LIN {X 0,Y 360.744,Z 841.948,A -85,B 0,C 180,E1 -13041.597,E2 -13041.597} C_VEL
LIN {X 0,Y 360.57,Z 846.721,A -85,B 0,C 180,E1 -13043.283,E2 -13043.283} C_VEL
LIN {X 0,Y 360.444,Z 850.328,A -85,B 0,C 180,E1 -13044.965,E2 -13044.965} C_VEL
LIN {X 0,Y 360.392,Z 852.877,A -85,B 0,C 180,E1 -13046.645,E2 -13046.645} C_VEL
LIN {X 0,Y 360.505,Z 854.049,A -85,B 0,C 180,E1 -13047.764,E2 -13047.764} C_VEL
LIN {X 0,Y 360.532,Z 854.752,A -85,B 0,C 180,E1 -13048.882,E2 -13048.882} C_VEL
LIN {X 0,Y 360.519,Z 855.046,A -85,B 0,C 180,E1 -13049.999,E2 -13049.999} C_VEL
LIN {X 0,Y 360.53,Z 854.935,A -85,B 0,C 180,E1 -13051.116,E2 -13051.116} C_VEL
LIN {X 0,Y 360.472,Z 854.395,A -85,B 0,C 180,E1 -13052.233,E2 -13052.233} C_VEL
LIN {X 0,Y 360.384,Z 853.407,A -85,B 0,C 180,E1 -13053.353,E2 -13053.353} C_VEL
LIN {X 0,Y 360.41,Z 852.013,A -85,B 0,C 180,E1 -13054.472,E2 -13054.472} C_VEL
LIN {X 0,Y 360.39,Z 849.445,A -85,B 0,C 180,E1 -13055.978,E2 -13055.978} C_VEL
LIN {X 0,Y 360.645,Z 845.108,A -85,B 0,C 180,E1 -13057.839,E2 -13057.839} C_VEL
LIN {X 0,Y 360.987,Z 839.985,A -85,B 0,C 180,E1 -13059.524,E2 -13059.524} C_VEL
LIN {X 0,Y 361.519,Z 833.569,A -85,B 0,C 180,E1 -13061.208,E2 -13061.208} C_VEL
LIN {X 0,Y 362.453,Z 825.598,A -85,B 0,C 180,E1 -13062.883,E2 -13062.883} C_VEL
LIN {X 0,Y 363.304,Z 817.472,A -85,B 0,C 180,E1 -13064.278,E2 -13064.278} C_VEL
LIN {X 0,Y 364.433,Z 806.509,A -85,B 0,C 180,E1 -13065.806,E2 -13065.806} C_VEL
LIN {X 0,Y 365.658,Z 795.285,A -85,B 0,C 180,E1 -13067.043,E2 -13067.043} C_VEL
LIN {X 0,Y 366.98,Z 782.593,A -85,B 0,C 180,E1 -13068.13,E2 -13068.13} C_VEL
LIN {X 0,Y 367.909,Z 771.311,A -85,B 0,C 180,E1 -13068.876,E2 -13068.876} C_VEL
LIN {X 0,Y 368.869,Z 757.948,A -85,B 0,C 180,E1 -13069.512,E2 -13069.512} C_VEL
LIN {X 0,Y 369.409,Z 745.082,A -85,B 0,C 180,E1 -13069.916,E2 -13069.916} C_VEL
LIN {X 0,Y 371,Z 678.071,A -85,B 0,C 180,E1 -13071.407,E2 -13071.407} C_VEL
LIN {X 0,Y 368.045,Z 656.105,A -85,B 0,C 180,E1 -13072.161,E2 -13072.161} C_VEL
LIN {X 0,Y 365.134,Z 639.929,A -85,B 0,C 180,E1 -13072.806,E2 -13072.806} C_VEL
LIN {X 0,Y 366.915,Z 623.577,A -85,B 0,C 180,E1 -13076.443,E2 -13076.443} C_VEL
LIN {X 0,Y 365.233,Z 614.506,A -85,B 0,C 180,E1 -13078.753,E2 -13078.753} C_VEL
LIN {X 0,Y 362.83,Z 604.307,A -85,B 0,C 180,E1 -13081.539,E2 -13081.539} C_VEL
LIN {X 0,Y 361.863,Z 600.413,A -85,B 0,C 180,E1 -13082.693,E2 -13082.693} C_VEL
LIN {X 0,Y 361.865,Z 600.411,A -85,B 0,C 180,E1 -13085.635,E2 -13085.635} C_VEL
LIN {X 0,Y 361.871,Z 600.411,A -85,B 0,C 180,E1 -13089.026,E2 -13089.026} C_VEL
LIN {X 0,Y 361.853,Z 600.414,A -85,B 0,C 180,E1 -13092.434,E2 -13092.434} C_VEL
LIN {X 0,Y 361.908,Z 600.407,A -85,B 0,C 180,E1 -13095.93,E2 -13095.93} C_VEL
LIN {X 0,Y 361.9,Z 600.405,A -85,B 0,C 180,E1 -13099.231,E2 -13099.231} C_VEL
LIN {X 0,Y 361.868,Z 600.406,A -85,B 0,C 180,E1 -13102.982,E2 -13102.982} C_VEL
LIN {X 0,Y 361.857,Z 600.409,A -85,B 0,C 180,E1 -13106.628,E2 -13106.628} C_VEL
LIN {X 0,Y 361.872,Z 600.405,A -85,B 0,C 180,E1 -13109.672,E2 -13109.672} C_VEL
LIN {X 0,Y 361.947,Z 600.394,A -85,B 0,C 180,E1 -13113.474,E2 -13113.474} C_VEL
LIN {X 0,Y 361.884,Z 600.404,A -85,B 0,C 180,E1 -13117.144,E2 -13117.144} C_VEL
LIN {X 0,Y 361.913,Z 600.405,A -85,B 0,C 180,E1 -13120.724,E2 -13120.724} C_VEL
LIN {X 0,Y 361.938,Z 600.402,A -85,B 0,C 180,E1 -13124.226,E2 -13124.226} C_VEL
LIN {X 0,Y 361.992,Z 600.395,A -85,B 0,C 180,E1 -13126.527,E2 -13126.527} C_VEL
LIN {X 0,Y 362.028,Z 600.388,A -85,B 0,C 180,E1 -13129.938,E2 -13129.938} C_VEL
LIN {X 0,Y 362.142,Z 600.375,A -85,B 0,C 180,E1 -13132.192,E2 -13132.192} C_VEL
LIN {X 0,Y 362.11,Z 600.379,A -85,B 0,C 180,E1 -13134.431,E2 -13134.431} C_VEL
LIN {X 0,Y 362.275,Z 600.359,A -85,B 0,C 180,E1 -13137.776,E2 -13137.776} C_VEL
LIN {X 0,Y 362.421,Z 600.343,A -85,B 0,C 180,E1 -13140,E2 -13140} C_VEL
LIN {X 0,Y 362.275,Z 600.359,A -85,B 0,C 180,E1 -13142.223,E2 -13142.223} C_VEL
LIN {X 0,Y 362.17,Z 600.377,A -85,B 0,C 180,E1 -13146.686,E2 -13146.686} C_VEL
LIN {X 0,Y 362.067,Z 600.387,A -85,B 0,C 180,E1 -13148.933,E2 -13148.933} C_VEL
LIN {X 0,Y 362.037,Z 600.45,A -85,B 0,C 180,E1 -13150.274,E2 -13150.274} C_VEL
LIN {X 0,Y 363.166,Z 605.77,A -85,B 0,C 180,E1 -13152.113,E2 -13152.113} C_VEL
LIN {X 0,Y 370.828,Z 623.781,A -85,B 0,C 180,E1 -13153.202,E2 -13153.202} C_VEL
LIN {X 0,Y 372.101,Z 628.288,A -85,B 0,C 180,E1 -13153.409,E2 -13153.409} C_VEL
LIN {X 0,Y 369.856,Z 712.137,A -85,B 0,C 180,E1 -13155.306,E2 -13155.306} C_VEL
LIN {X 0,Y 369.281,Z 725.643,A -85,B 0,C 180,E1 -13155.842,E2 -13155.842} C_VEL
LIN {X 0,Y 368.533,Z 737.945,A -85,B 0,C 180,E1 -13156.55,E2 -13156.55} C_VEL
LIN {X 0,Y 367.596,Z 750.201,A -85,B 0,C 180,E1 -13157.507,E2 -13157.507} C_VEL
LIN {X 0,Y 366.603,Z 761.038,A -85,B 0,C 180,E1 -13158.585,E2 -13158.585} C_VEL
LIN {X 0,Y 365.372,Z 771.583,A -85,B 0,C 180,E1 -13159.891,E2 -13159.891} C_VEL
LIN {X 0,Y 364.418,Z 780.085,A -85,B 0,C 180,E1 -13161.199,E2 -13161.199} C_VEL
LIN {X 0,Y 363.405,Z 788.357,A -85,B 0,C 180,E1 -13162.755,E2 -13162.755} C_VEL
LIN {X 0,Y 362.543,Z 795.203,A -85,B 0,C 180,E1 -13164.345,E2 -13164.345} C_VEL
LIN {X 0,Y 361.987,Z 800.581,A -85,B 0,C 180,E1 -13165.902,E2 -13165.902} C_VEL
LIN {X 0,Y 361.349,Z 805.776,A -85,B 0,C 180,E1 -13167.826,E2 -13167.826} C_VEL
LIN {X 0,Y 360.895,Z 809.537,A -85,B 0,C 180,E1 -13169.774,E2 -13169.774} C_VEL
LIN {X 0,Y 360.552,Z 812.009,A -85,B 0,C 180,E1 -13171.755,E2 -13171.755} C_VEL
LIN {X 0,Y 360.407,Z 812.942,A -85,B 0,C 180,E1 -13173.093,E2 -13173.093} C_VEL
LIN {X 0,Y 360.341,Z 813.24,A -85,B 0,C 180,E1 -13175.002,E2 -13175.002} C_VEL
LIN {X 0,Y 360.356,Z 812.132,A -85,B 0,C 180,E1 -13177.199,E2 -13177.199} C_VEL
LIN {X 0,Y 360.585,Z 809.482,A -85,B 0,C 180,E1 -13179.344,E2 -13179.344} C_VEL
LIN {X 0,Y 360.805,Z 807.257,A -85,B 0,C 180,E1 -13180.567,E2 -13180.567} C_VEL
LIN {X 0,Y 361.082,Z 803.145,A -85,B 0,C 180,E1 -13182.303,E2 -13182.303} C_VEL
LIN {X 0,Y 361.548,Z 797.876,A -85,B 0,C 180,E1 -13184.011,E2 -13184.011} C_VEL
LIN {X 0,Y 362.233,Z 790.465,A -85,B 0,C 180,E1 -13185.879,E2 -13185.879} C_VEL
LIN {X 0,Y 363.055,Z 782.045,A -85,B 0,C 180,E1 -13187.563,E2 -13187.563} C_VEL
LIN {X 0,Y 363.939,Z 772.774,A -85,B 0,C 180,E1 -13189.051,E2 -13189.051} C_VEL
LIN {X 0,Y 364.878,Z 762.379,A -85,B 0,C 180,E1 -13190.394,E2 -13190.394} C_VEL
LIN {X 0,Y 365.792,Z 751.243,A -85,B 0,C 180,E1 -13191.55,E2 -13191.55} C_VEL
LIN {X 0,Y 366.608,Z 739.771,A -85,B 0,C 180,E1 -13192.481,E2 -13192.481} C_VEL
LIN {X 0,Y 367.297,Z 726.855,A -85,B 0,C 180,E1 -13193.278,E2 -13193.278} C_VEL
LIN {X 0,Y 367.781,Z 714.021,A -85,B 0,C 180,E1 -13193.836,E2 -13193.836} C_VEL
LIN {X 0,Y 368.178,Z 697.844,A -85,B 0,C 180,E1 -13194.249,E2 -13194.249} C_VEL
LIN {X 0,Y 369.593,Z 625.625,A -85,B 0,C 180,E1 -13195.797,E2 -13195.797} C_VEL
LIN {X 0,Y 367.76,Z 618.455,A -85,B 0,C 180,E1 -13196.058,E2 -13196.058} C_VEL
LIN {X 0,Y 362.366,Z 602.699,A -85,B 0,C 180,E1 -13196.733,E2 -13196.733} C_VEL
LIN {X 0,Y 361.879,Z 600.408,A -85,B 0,C 180,E1 -13197.473,E2 -13197.473} C_VEL
LIN {X 0,Y 361.896,Z 600.402,A -85,B 0,C 180,E1 -13200.956,E2 -13200.956} C_VEL
LIN {X 0,Y 361.951,Z 600.396,A -85,B 0,C 180,E1 -13203.476,E2 -13203.476} C_VEL
LIN {X 0,Y 361.891,Z 600.402,A -85,B 0,C 180,E1 -13207.146,E2 -13207.146} C_VEL
LIN {X 0,Y 361.926,Z 600.399,A -85,B 0,C 180,E1 -13210.726,E2 -13210.726} C_VEL
LIN {X 0,Y 361.945,Z 600.402,A -85,B 0,C 180,E1 -13214.227,E2 -13214.227} C_VEL
LIN {X 0,Y 361.999,Z 600.393,A -85,B 0,C 180,E1 -13216.529,E2 -13216.529} C_VEL
LIN {X 0,Y 362.036,Z 600.387,A -85,B 0,C 180,E1 -13219.939,E2 -13219.939} C_VEL
LIN {X 0,Y 362.152,Z 600.374,A -85,B 0,C 180,E1 -13222.194,E2 -13222.194} C_VEL
LIN {X 0,Y 362.119,Z 600.381,A -85,B 0,C 180,E1 -13224.433,E2 -13224.433} C_VEL
LIN {X 0,Y 362.284,Z 600.354,A -85,B 0,C 180,E1 -13227.778,E2 -13227.778} C_VEL
LIN {X 0,Y 362.427,Z 600.337,A -85,B 0,C 180,E1 -13230.001,E2 -13230.001} C_VEL
LIN {X 0,Y 362.284,Z 600.356,A -85,B 0,C 180,E1 -13232.225,E2 -13232.225} C_VEL
LIN {X 0,Y 362.174,Z 600.374,A -85,B 0,C 180,E1 -13236.687,E2 -13236.687} C_VEL
LIN {X 0,Y 362.034,Z 600.385,A -85,B 0,C 180,E1 -13239.616,E2 -13239.616} C_VEL
LIN {X 0,Y 361.354,Z 600.474,A -85,B 0,C 180,E1 -13240.544,E2 -13240.544} C_VEL
LIN {X 0,Y 358.482,Z 600.827,A -85,B 0,C 180,E1 -13242.053,E2 -13242.053} C_VEL
LIN {X 0,Y 356.053,Z 601.131,A -85,B 0,C 180,E1 -13243.274,E2 -13243.274} C_VEL
LIN {X 0,Y 355.008,Z 601.261,A -85,B 0,C 180,E1 -13244.219,E2 -13244.219} C_VEL
LIN {X 0,Y 354.921,Z 601.273,A -85,B 0,C 180,E1 -13244.539,E2 -13244.539} C_VEL
LIN {X 0,Y 354.904,Z 601.275,A -85,B 0,C 180,E1 -13248.473,E2 -13248.473} C_VEL
LIN {X 0,Y 354.838,Z 601.281,A -85,B 0,C 180,E1 -13252.107,E2 -13252.107} C_VEL
LIN {X 0,Y 354.902,Z 601.273,A -85,B 0,C 180,E1 -13255.828,E2 -13255.828} C_VEL
LIN {X 0,Y 354.821,Z 601.284,A -85,B 0,C 180,E1 -13259.683,E2 -13259.683} C_VEL
LIN {X 0,Y 354.81,Z 601.286,A -85,B 0,C 180,E1 -13263.703,E2 -13263.703} C_VEL
LIN {X 0,Y 354.801,Z 601.286,A -85,B 0,C 180,E1 -13266.46,E2 -13266.46} C_VEL
LIN {X 0,Y 354.828,Z 601.287,A -85,B 0,C 180,E1 -13269.424,E2 -13269.424} C_VEL
LIN {X 0,Y 354.792,Z 601.289,A -85,B 0,C 180,E1 -13272.868,E2 -13272.868} C_VEL
LIN {X 0,Y 354.784,Z 601.288,A -85,B 0,C 180,E1 -13276.106,E2 -13276.106} C_VEL
LIN {X 0,Y 354.792,Z 601.29,A -85,B 0,C 180,E1 -13279.18,E2 -13279.18} C_VEL
LIN {X 0,Y 354.811,Z 601.284,A -85,B 0,C 180,E1 -13282.403,E2 -13282.403} C_VEL
LIN {X 0,Y 354.817,Z 601.285,A -85,B 0,C 180,E1 -13284.941,E2 -13284.941} C_VEL
LIN {X 0,Y 354.8,Z 601.286,A -85,B 0,C 180,E1 -13288.405,E2 -13288.405} C_VEL
LIN {X 0,Y 354.856,Z 601.285,A -85,B 0,C 180,E1 -13291.62,E2 -13291.62} C_VEL
LIN {X 0,Y 354.904,Z 601.275,A -85,B 0,C 180,E1 -13294.173,E2 -13294.173} C_VEL
LIN {X 0,Y 354.821,Z 601.289,A -85,B 0,C 180,E1 -13297.893,E2 -13297.893} C_VEL
LIN {X 0,Y 354.928,Z 601.276,A -85,B 0,C 180,E1 -13301.892,E2 -13301.892} C_VEL
LIN {X 0,Y 354.949,Z 601.273,A -85,B 0,C 180,E1 -13305.981,E2 -13305.981} C_VEL
LIN {X 0,Y 354.983,Z 601.266,A -85,B 0,C 180,E1 -13309.736,E2 -13309.736} C_VEL
LIN {X 0,Y 355.13,Z 601.245,A -85,B 0,C 180,E1 -13313.181,E2 -13313.181} C_VEL
LIN {X 0,Y 355.249,Z 601.232,A -85,B 0,C 180,E1 -13317.733,E2 -13317.733} C_VEL
LIN {X 0,Y 355.402,Z 601.215,A -85,B 0,C 180,E1 -13320,E2 -13320} C_VEL
LIN {X 0,Y 355.249,Z 601.236,A -85,B 0,C 180,E1 -13322.268,E2 -13322.268} C_VEL
LIN {X 0,Y 355.132,Z 601.246,A -85,B 0,C 180,E1 -13326.819,E2 -13326.819} C_VEL
LIN {X 0,Y 354.984,Z 601.268,A -85,B 0,C 180,E1 -13330.264,E2 -13330.264} C_VEL
LIN {X 0,Y 354.949,Z 601.269,A -85,B 0,C 180,E1 -13334.019,E2 -13334.019} C_VEL
LIN {X 0,Y 354.896,Z 601.276,A -85,B 0,C 180,E1 -13338.092,E2 -13338.092} C_VEL
LIN {X 0,Y 354.823,Z 601.285,A -85,B 0,C 180,E1 -13342.107,E2 -13342.107} C_VEL
LIN {X 0,Y 354.905,Z 601.273,A -85,B 0,C 180,E1 -13345.827,E2 -13345.827} C_VEL
LIN {X 0,Y 354.86,Z 601.278,A -85,B 0,C 180,E1 -13349.678,E2 -13349.678} C_VEL
LIN {X 0,Y 354.812,Z 601.284,A -85,B 0,C 180,E1 -13353.702,E2 -13353.702} C_VEL
LIN {X 0,Y 354.803,Z 601.288,A -85,B 0,C 180,E1 -13356.459,E2 -13356.459} C_VEL
LIN {X 0,Y 354.83,Z 601.284,A -85,B 0,C 180,E1 -13359.423,E2 -13359.423} C_VEL
LIN {X 0,Y 354.794,Z 601.292,A -85,B 0,C 180,E1 -13362.867,E2 -13362.867} C_VEL
LIN {X 0,Y 354.78,Z 601.288,A -85,B 0,C 180,E1 -13366.104,E2 -13366.104} C_VEL
LIN {X 0,Y 354.794,Z 601.292,A -85,B 0,C 180,E1 -13369.179,E2 -13369.179} C_VEL
LIN {X 0,Y 354.813,Z 601.284,A -85,B 0,C 180,E1 -13372.402,E2 -13372.402} C_VEL
LIN {X 0,Y 354.817,Z 601.287,A -85,B 0,C 180,E1 -13374.94,E2 -13374.94} C_VEL
LIN {X 0,Y 354.846,Z 601.486,A -85,B 0,C 180,E1 -13378.51,E2 -13378.51} C_VEL
LIN {X 0,Y 357.812,Z 615.009,A -85,B 0,C 180,E1 -13381.874,E2 -13381.874} C_VEL
LIN {X 0,Y 359.157,Z 622.011,A -85,B 0,C 180,E1 -13383.553,E2 -13383.553} C_VEL
LIN {X 0,Y 358.818,Z 627.547,A -85,B 0,C 180,E1 -13384.784,E2 -13384.784} C_VEL
LIN {X 0,Y 357.382,Z 642.401,A -85,B 0,C 180,E1 -13387.999,E2 -13387.999} C_VEL
LIN {X 0,Y 362.247,Z 679.252,A -85,B 0,C 180,E1 -13389.12,E2 -13389.12} C_VEL
LIN {X 0,Y 360.747,Z 751.541,A -85,B 0,C 180,E1 -13390.732,E2 -13390.732} C_VEL
LIN {X 0,Y 360.082,Z 765.709,A -85,B 0,C 180,E1 -13391.286,E2 -13391.286} C_VEL
LIN {X 0,Y 359.204,Z 777.806,A -85,B 0,C 180,E1 -13391.977,E2 -13391.977} C_VEL
LIN {X 0,Y 358.25,Z 789.595,A -85,B 0,C 180,E1 -13392.885,E2 -13392.885} C_VEL
LIN {X 0,Y 357.184,Z 801.01,A -85,B 0,C 180,E1 -13394.009,E2 -13394.009} C_VEL
LIN {X 0,Y 356.313,Z 811.37,A -85,B 0,C 180,E1 -13395.291,E2 -13395.291} C_VEL
LIN {X 0,Y 355.304,Z 821.45,A -85,B 0,C 180,E1 -13396.85,E2 -13396.85} C_VEL
LIN {X 0,Y 354.457,Z 830.346,A -85,B 0,C 180,E1 -13398.563,E2 -13398.563} C_VEL
LIN {X 0,Y 353.935,Z 837.426,A -85,B 0,C 180,E1 -13400.282,E2 -13400.282} C_VEL
LIN {X 0,Y 353.572,Z 843.076,A -85,B 0,C 180,E1 -13402.001,E2 -13402.001} C_VEL
LIN {X 0,Y 353.391,Z 847.926,A -85,B 0,C 180,E1 -13403.918,E2 -13403.918} C_VEL
LIN {X 0,Y 353.383,Z 850.777,A -85,B 0,C 180,E1 -13405.436,E2 -13405.436} C_VEL
LIN {X 0,Y 353.31,Z 852.391,A -85,B 0,C 180,E1 -13406.578,E2 -13406.578} C_VEL
LIN {X 0,Y 353.406,Z 853.588,A -85,B 0,C 180,E1 -13407.719,E2 -13407.719} C_VEL
LIN {X 0,Y 353.468,Z 854.314,A -85,B 0,C 180,E1 -13408.859,E2 -13408.859} C_VEL
LIN {X 0,Y 353.454,Z 854.621,A -85,B 0,C 180,E1 -13409.999,E2 -13409.999} C_VEL
LIN {X 0,Y 353.465,Z 854.523,A -85,B 0,C 180,E1 -13411.138,E2 -13411.138} C_VEL
LIN {X 0,Y 353.372,Z 854.005,A -85,B 0,C 180,E1 -13412.278,E2 -13412.278} C_VEL
LIN {X 0,Y 353.301,Z 853.031,A -85,B 0,C 180,E1 -13413.42,E2 -13413.42} C_VEL
LIN {X 0,Y 353.318,Z 851.652,A -85,B 0,C 180,E1 -13414.562,E2 -13414.562} C_VEL
LIN {X 0,Y 353.314,Z 849.381,A -85,B 0,C 180,E1 -13415.964,E2 -13415.964} C_VEL
LIN {X 0,Y 353.57,Z 844.818,A -85,B 0,C 180,E1 -13417.997,E2 -13417.997} C_VEL
LIN {X 0,Y 353.961,Z 839.729,A -85,B 0,C 180,E1 -13419.715,E2 -13419.715} C_VEL
LIN {X 0,Y 354.525,Z 833.342,A -85,B 0,C 180,E1 -13421.433,E2 -13421.433} C_VEL
LIN {X 0,Y 355.515,Z 825.43,A -85,B 0,C 180,E1 -13423.139,E2 -13423.139} C_VEL
LIN {X 0,Y 356.412,Z 817.35,A -85,B 0,C 180,E1 -13424.56,E2 -13424.56} C_VEL
LIN {X 0,Y 357.464,Z 807.528,A -85,B 0,C 180,E1 -13425.976,E2 -13425.976} C_VEL
LIN {X 0,Y 358.721,Z 796.729,A -85,B 0,C 180,E1 -13427.236,E2 -13427.236} C_VEL
LIN {X 0,Y 359.912,Z 786.348,A -85,B 0,C 180,E1 -13428.204,E2 -13428.204} C_VEL
LIN {X 0,Y 360.916,Z 775.17,A -85,B 0,C 180,E1 -13429.035,E2 -13429.035} C_VEL
LIN {X 0,Y 362.107,Z 761.372,A -85,B 0,C 180,E1 -13429.78,E2 -13429.78} C_VEL
LIN {X 0,Y 362.846,Z 748.469,A -85,B 0,C 180,E1 -13430.255,E2 -13430.255} C_VEL
LIN {X 0,Y 364.545,Z 678.837,A -85,B 0,C 180,E1 -13431.856,E2 -13431.856} C_VEL
LIN {X 0,Y 361.805,Z 658.147,A -85,B 0,C 180,E1 -13432.589,E2 -13432.589} C_VEL
LIN {X 0,Y 358.687,Z 641.12,A -85,B 0,C 180,E1 -13433.285,E2 -13433.285} C_VEL
LIN {X 0,Y 358.392,Z 639.424,A -85,B 0,C 180,E1 -13433.367,E2 -13433.367} C_VEL
LIN {X 0,Y 359.916,Z 626.7,A -85,B 0,C 180,E1 -13436.254,E2 -13436.254} C_VEL
LIN {X 0,Y 359.825,Z 623.617,A -85,B 0,C 180,E1 -13437.006,E2 -13437.006} C_VEL
LIN {X 0,Y 358.052,Z 614.621,A -85,B 0,C 180,E1 -13439.386,E2 -13439.386} C_VEL
LIN {X 0,Y 355.344,Z 603.336,A -85,B 0,C 180,E1 -13442.611,E2 -13442.611} C_VEL
LIN {X 0,Y 354.833,Z 601.289,A -85,B 0,C 180,E1 -13443.255,E2 -13443.255} C_VEL
LIN {X 0,Y 354.796,Z 601.292,A -85,B 0,C 180,E1 -13446.458,E2 -13446.458} C_VEL
LIN {X 0,Y 354.82,Z 601.289,A -85,B 0,C 180,E1 -13449.422,E2 -13449.422} C_VEL
LIN {X 0,Y 354.803,Z 601.292,A -85,B 0,C 180,E1 -13452.869,E2 -13452.869} C_VEL
LIN {X 0,Y 354.847,Z 601.286,A -85,B 0,C 180,E1 -13456.116,E2 -13456.116} C_VEL
LIN {X 0,Y 354.851,Z 601.283,A -85,B 0,C 180,E1 -13459.187,E2 -13459.187} C_VEL
LIN {X 0,Y 354.807,Z 601.291,A -85,B 0,C 180,E1 -13462.4,E2 -13462.4} C_VEL
LIN {X 0,Y 354.806,Z 601.287,A -85,B 0,C 180,E1 -13464.94,E2 -13464.94} C_VEL
LIN {X 0,Y 354.81,Z 601.284,A -85,B 0,C 180,E1 -13468.398,E2 -13468.398} C_VEL
LIN {X 0,Y 354.849,Z 601.276,A -85,B 0,C 180,E1 -13471.619,E2 -13471.619} C_VEL
LIN {X 0,Y 354.892,Z 601.273,A -85,B 0,C 180,E1 -13474.172,E2 -13474.172} C_VEL
LIN {X 0,Y 354.828,Z 601.284,A -85,B 0,C 180,E1 -13477.893,E2 -13477.893} C_VEL
LIN {X 0,Y 354.915,Z 601.275,A -85,B 0,C 180,E1 -13481.891,E2 -13481.891} C_VEL
LIN {X 0,Y 354.935,Z 601.271,A -85,B 0,C 180,E1 -13485.98,E2 -13485.98} C_VEL
LIN {X 0,Y 354.974,Z 601.268,A -85,B 0,C 180,E1 -13489.736,E2 -13489.736} C_VEL
LIN {X 0,Y 355.105,Z 601.252,A -85,B 0,C 180,E1 -13492.037,E2 -13492.037} C_VEL
LIN {X 0,Y 355.084,Z 601.254,A -85,B 0,C 180,E1 -13494.32,E2 -13494.32} C_VEL
LIN {X 0,Y 355.238,Z 601.235,A -85,B 0,C 180,E1 -13497.732,E2 -13497.732} C_VEL
LIN {X 0,Y 355.391,Z 601.218,A -85,B 0,C 180,E1 -13500,E2 -13500} C_VEL
LIN {X 0,Y 355.238,Z 601.236,A -85,B 0,C 180,E1 -13502.268,E2 -13502.268} C_VEL
LIN {X 0,Y 355.135,Z 601.252,A -85,B 0,C 180,E1 -13506.819,E2 -13506.819} C_VEL
LIN {X 0,Y 355.018,Z 601.397,A -85,B 0,C 180,E1 -13509.759,E2 -13509.759} C_VEL
LIN {X 0,Y 356.161,Z 606.616,A -85,B 0,C 180,E1 -13511.543,E2 -13511.543} C_VEL
LIN {X 0,Y 363.651,Z 623.662,A -85,B 0,C 180,E1 -13512.631,E2 -13512.631} C_VEL
LIN {X 0,Y 365.624,Z 628.879,A -85,B 0,C 180,E1 -13512.926,E2 -13512.926} C_VEL
LIN {X 0,Y 363.347,Z 712.775,A -85,B 0,C 180,E1 -13514.878,E2 -13514.878} C_VEL
LIN {X 0,Y 362.76,Z 725.747,A -85,B 0,C 180,E1 -13515.4,E2 -13515.4} C_VEL
LIN {X 0,Y 361.978,Z 738.328,A -85,B 0,C 180,E1 -13516.134,E2 -13516.134} C_VEL
LIN {X 0,Y 361.032,Z 750.261,A -85,B 0,C 180,E1 -13517.077,E2 -13517.077} C_VEL
LIN {X 0,Y 359.938,Z 761.45,A -85,B 0,C 180,E1 -13518.204,E2 -13518.204} C_VEL
LIN {X 0,Y 358.715,Z 771.442,A -85,B 0,C 180,E1 -13519.455,E2 -13519.455} C_VEL
LIN {X 0,Y 357.493,Z 781.393,A -85,B 0,C 180,E1 -13521.025,E2 -13521.025} C_VEL
LIN {X 0,Y 356.415,Z 789.739,A -85,B 0,C 180,E1 -13522.659,E2 -13522.659} C_VEL
LIN {X 0,Y 355.565,Z 796.159,A -85,B 0,C 180,E1 -13524.213,E2 -13524.213} C_VEL
LIN {X 0,Y 354.967,Z 801.507,A -85,B 0,C 180,E1 -13525.822,E2 -13525.822} C_VEL
LIN {X 0,Y 354.303,Z 806.553,A -85,B 0,C 180,E1 -13527.785,E2 -13527.785} C_VEL
LIN {X 0,Y 353.821,Z 810.222,A -85,B 0,C 180,E1 -13529.774,E2 -13529.774} C_VEL
LIN {X 0,Y 353.535,Z 812.097,A -85,B 0,C 180,E1 -13531.265,E2 -13531.265} C_VEL
LIN {X 0,Y 353.311,Z 813.5,A -85,B 0,C 180,E1 -13533.339,E2 -13533.339} C_VEL
LIN {X 0,Y 353.239,Z 813.586,A -85,B 0,C 180,E1 -13535.343,E2 -13535.343} C_VEL
LIN {X 0,Y 353.291,Z 812.474,A -85,B 0,C 180,E1 -13537.28,E2 -13537.28} C_VEL
LIN {X 0,Y 353.528,Z 809.674,A -85,B 0,C 180,E1 -13539.505,E2 -13539.505} C_VEL
LIN {X 0,Y 353.933,Z 805.31,A -85,B 0,C 180,E1 -13541.697,E2 -13541.697} C_VEL
LIN {X 0,Y 354.353,Z 799.916,A -85,B 0,C 180,E1 -13543.625,E2 -13543.625} C_VEL
LIN {X 0,Y 355.006,Z 793.3,A -85,B 0,C 180,E1 -13545.454,E2 -13545.454} C_VEL
LIN {X 0,Y 355.755,Z 785.33,A -85,B 0,C 180,E1 -13547.205,E2 -13547.205} C_VEL
LIN {X 0,Y 356.682,Z 776.454,A -85,B 0,C 180,E1 -13548.758,E2 -13548.758} C_VEL
LIN {X 0,Y 357.715,Z 766.008,A -85,B 0,C 180,E1 -13550.236,E2 -13550.236} C_VEL
LIN {X 0,Y 358.591,Z 755.652,A -85,B 0,C 180,E1 -13551.413,E2 -13551.413} C_VEL
LIN {X 0,Y 359.517,Z 743.5,A -85,B 0,C 180,E1 -13552.501,E2 -13552.501} C_VEL
LIN {X 0,Y 360.23,Z 731.788,A -85,B 0,C 180,E1 -13553.312,E2 -13553.312} C_VEL
LIN {X 0,Y 360.776,Z 718.94,A -85,B 0,C 180,E1 -13553.961,E2 -13553.961} C_VEL
LIN {X 0,Y 361.241,Z 704.964,A -85,B 0,C 180,E1 -13554.409,E2 -13554.409} C_VEL
LIN {X 0,Y 362.863,Z 626.732,A -85,B 0,C 180,E1 -13556.129,E2 -13556.129} C_VEL
LIN {X 0,Y 361.209,Z 620.522,A -85,B 0,C 180,E1 -13556.362,E2 -13556.362} C_VEL
LIN {X 0,Y 355.177,Z 603.1,A -85,B 0,C 180,E1 -13557.119,E2 -13557.119} C_VEL
LIN {X 0,Y 354.837,Z 601.286,A -85,B 0,C 180,E1 -13557.731,E2 -13557.731} C_VEL
LIN {X 0,Y 354.843,Z 601.283,A -85,B 0,C 180,E1 -13561.62,E2 -13561.62} C_VEL
LIN {X 0,Y 354.896,Z 601.279,A -85,B 0,C 180,E1 -13564.174,E2 -13564.174} C_VEL
LIN {X 0,Y 354.837,Z 601.285,A -85,B 0,C 180,E1 -13567.896,E2 -13567.896} C_VEL
LIN {X 0,Y 354.922,Z 601.274,A -85,B 0,C 180,E1 -13571.892,E2 -13571.892} C_VEL
LIN {X 0,Y 354.942,Z 601.271,A -85,B 0,C 180,E1 -13575.982,E2 -13575.982} C_VEL
LIN {X 0,Y 354.982,Z 601.264,A -85,B 0,C 180,E1 -13579.737,E2 -13579.737} C_VEL
LIN {X 0,Y 355.115,Z 601.249,A -85,B 0,C 180,E1 -13582.038,E2 -13582.038} C_VEL
LIN {X 0,Y 355.093,Z 601.254,A -85,B 0,C 180,E1 -13584.322,E2 -13584.322} C_VEL
LIN {X 0,Y 355.247,Z 601.23,A -85,B 0,C 180,E1 -13587.734,E2 -13587.734} C_VEL
LIN {X 0,Y 355.397,Z 601.213,A -85,B 0,C 180,E1 -13590.001,E2 -13590.001} C_VEL
LIN {X 0,Y 355.247,Z 601.233,A -85,B 0,C 180,E1 -13592.269,E2 -13592.269} C_VEL
LIN {X 0,Y 355.14,Z 601.248,A -85,B 0,C 180,E1 -13596.82,E2 -13596.82} C_VEL
LIN {X 0,Y 354.984,Z 601.263,A -85,B 0,C 180,E1 -13599.609,E2 -13599.609} C_VEL
LIN {X 0,Y 354.954,Z 601.266,A -85,B 0,C 180,E1 -13603.746,E2 -13603.746} C_VEL
LIN {X 0,Y 354.921,Z 601.273,A -85,B 0,C 180,E1 -13604.539,E2 -13604.539} C_VEL
LIN {X 0,Y 354.246,Z 601.362,A -85,B 0,C 180,E1 -13605.486,E2 -13605.486} C_VEL
LIN {X 0,Y 351.378,Z 601.721,A -85,B 0,C 180,E1 -13607.027,E2 -13607.027} C_VEL
LIN {X 0,Y 348.948,Z 602.02,A -85,B 0,C 180,E1 -13608.274,E2 -13608.274} C_VEL
LIN {X 0,Y 347.9,Z 602.149,A -85,B 0,C 180,E1 -13609.24,E2 -13609.24} C_VEL
LIN {X 0,Y 347.812,Z 602.157,A -85,B 0,C 180,E1 -13609.567,E2 -13609.567} C_VEL
LIN {X 0,Y 347.777,Z 602.163,A -85,B 0,C 180,E1 -13612.58,E2 -13612.58} C_VEL
LIN {X 0,Y 347.816,Z 602.161,A -85,B 0,C 180,E1 -13615.109,E2 -13615.109} C_VEL
LIN {X 0,Y 347.811,Z 602.157,A -85,B 0,C 180,E1 -13617.695,E2 -13617.695} C_VEL
LIN {X 0,Y 347.753,Z 602.164,A -85,B 0,C 180,E1 -13620.349,E2 -13620.349} C_VEL
LIN {X 0,Y 347.752,Z 602.164,A -85,B 0,C 180,E1 -13624.045,E2 -13624.045} C_VEL
LIN {X 0,Y 347.766,Z 602.168,A -85,B 0,C 180,E1 -13627.322,E2 -13627.322} C_VEL
LIN {X 0,Y 347.736,Z 602.166,A -85,B 0,C 180,E1 -13630.298,E2 -13630.298} C_VEL
LIN {X 0,Y 347.727,Z 602.173,A -85,B 0,C 180,E1 -13633.409,E2 -13633.409} C_VEL
LIN {X 0,Y 347.732,Z 602.167,A -85,B 0,C 180,E1 -13636.687,E2 -13636.687} C_VEL
LIN {X 0,Y 347.752,Z 602.164,A -85,B 0,C 180,E1 -13640.174,E2 -13640.174} C_VEL
LIN {X 0,Y 347.766,Z 602.162,A -85,B 0,C 180,E1 -13642.68,E2 -13642.68} C_VEL
LIN {X 0,Y 347.753,Z 602.166,A -85,B 0,C 180,E1 -13645.957,E2 -13645.957} C_VEL
LIN {X 0,Y 347.769,Z 602.168,A -85,B 0,C 180,E1 -13649.654,E2 -13649.654} C_VEL
LIN {X 0,Y 347.857,Z 602.151,A -85,B 0,C 180,E1 -13652.745,E2 -13652.745} C_VEL
LIN {X 0,Y 347.79,Z 602.161,A -85,B 0,C 180,E1 -13656.162,E2 -13656.162} C_VEL
LIN {X 0,Y 347.814,Z 602.162,A -85,B 0,C 180,E1 -13659.91,E2 -13659.91} C_VEL
LIN {X 0,Y 347.872,Z 602.15,A -85,B 0,C 180,E1 -13662.36,E2 -13662.36} C_VEL
LIN {X 0,Y 347.903,Z 602.151,A -85,B 0,C 180,E1 -13665.971,E2 -13665.971} C_VEL
LIN {X 0,Y 347.934,Z 602.143,A -85,B 0,C 180,E1 -13669.526,E2 -13669.526} C_VEL
LIN {X 0,Y 348.097,Z 602.121,A -85,B 0,C 180,E1 -13673.042,E2 -13673.042} C_VEL
LIN {X 0,Y 348.212,Z 602.108,A -85,B 0,C 180,E1 -13677.687,E2 -13677.687} C_VEL
LIN {X 0,Y 348.351,Z 602.094,A -85,B 0,C 180,E1 -13680,E2 -13680} C_VEL
LIN {X 0,Y 348.212,Z 602.112,A -85,B 0,C 180,E1 -13682.314,E2 -13682.314} C_VEL
LIN {X 0,Y 348.098,Z 602.121,A -85,B 0,C 180,E1 -13686.958,E2 -13686.958} C_VEL
LIN {X 0,Y 347.934,Z 602.147,A -85,B 0,C 180,E1 -13690.474,E2 -13690.474} C_VEL
LIN {X 0,Y 347.905,Z 602.148,A -85,B 0,C 180,E1 -13694.15,E2 -13694.15} C_VEL
LIN {X 0,Y 347.835,Z 602.157,A -85,B 0,C 180,E1 -13698.259,E2 -13698.259} C_VEL
LIN {X 0,Y 347.774,Z 602.161,A -85,B 0,C 180,E1 -13701.626,E2 -13701.626} C_VEL
LIN {X 0,Y 347.817,Z 602.157,A -85,B 0,C 180,E1 -13705.108,E2 -13705.108} C_VEL
LIN {X 0,Y 347.817,Z 602.156,A -85,B 0,C 180,E1 -13707.694,E2 -13707.694} C_VEL
LIN {X 0,Y 347.77,Z 602.164,A -85,B 0,C 180,E1 -13710.346,E2 -13710.346} C_VEL
LIN {X 0,Y 347.75,Z 602.167,A -85,B 0,C 180,E1 -13714.464,E2 -13714.464} C_VEL
LIN {X 0,Y 347.779,Z 602.16,A -85,B 0,C 180,E1 -13717.988,E2 -13717.988} C_VEL
LIN {X 0,Y 347.756,Z 602.163,A -85,B 0,C 180,E1 -13721.83,E2 -13721.83} C_VEL
LIN {X 0,Y 347.772,Z 602.168,A -85,B 0,C 180,E1 -13725.016,E2 -13725.016} C_VEL
LIN {X 0,Y 347.756,Z 602.164,A -85,B 0,C 180,E1 -13728.397,E2 -13728.397} C_VEL
LIN {X 0,Y 347.779,Z 602.16,A -85,B 0,C 180,E1 -13732.011,E2 -13732.011} C_VEL
LIN {X 0,Y 347.75,Z 602.169,A -85,B 0,C 180,E1 -13735.535,E2 -13735.535} C_VEL
LIN {X 0,Y 347.796,Z 602.347,A -85,B 0,C 180,E1 -13738.191,E2 -13738.191} C_VEL
LIN {X 0,Y 350.737,Z 615.766,A -85,B 0,C 180,E1 -13741.604,E2 -13741.604} C_VEL
LIN {X 0,Y 352.259,Z 624.266,A -85,B 0,C 180,E1 -13743.677,E2 -13743.677} C_VEL
LIN {X 0,Y 350.651,Z 640.143,A -85,B 0,C 180,E1 -13747.216,E2 -13747.216} C_VEL
LIN {X 0,Y 350.48,Z 641.887,A -85,B 0,C 180,E1 -13747.603,E2 -13747.603} C_VEL
LIN {X 0,Y 355.448,Z 679.263,A -85,B 0,C 180,E1 -13748.776,E2 -13748.776} C_VEL
LIN {X 0,Y 353.938,Z 751.088,A -85,B 0,C 180,E1 -13750.421,E2 -13750.421} C_VEL
LIN {X 0,Y 353.255,Z 765.256,A -85,B 0,C 180,E1 -13750.986,E2 -13750.986} C_VEL
LIN {X 0,Y 352.338,Z 777.36,A -85,B 0,C 180,E1 -13751.689,E2 -13751.689} C_VEL
LIN {X 0,Y 351.28,Z 789.953,A -85,B 0,C 180,E1 -13752.685,E2 -13752.685} C_VEL
LIN {X 0,Y 350.177,Z 801.234,A -85,B 0,C 180,E1 -13753.83,E2 -13753.83} C_VEL
LIN {X 0,Y 349.294,Z 811.456,A -85,B 0,C 180,E1 -13755.138,E2 -13755.138} C_VEL
LIN {X 0,Y 348.334,Z 820.631,A -85,B 0,C 180,E1 -13756.583,E2 -13756.583} C_VEL
LIN {X 0,Y 347.472,Z 829.613,A -85,B 0,C 180,E1 -13758.33,E2 -13758.33} C_VEL
LIN {X 0,Y 346.888,Z 836.774,A -85,B 0,C 180,E1 -13760.082,E2 -13760.082} C_VEL
LIN {X 0,Y 346.517,Z 842.477,A -85,B 0,C 180,E1 -13761.837,E2 -13761.837} C_VEL
LIN {X 0,Y 346.347,Z 847.06,A -85,B 0,C 180,E1 -13763.649,E2 -13763.649} C_VEL
LIN {X 0,Y 346.293,Z 850.263,A -85,B 0,C 180,E1 -13765.342,E2 -13765.342} C_VEL
LIN {X 0,Y 346.232,Z 851.895,A -85,B 0,C 180,E1 -13766.508,E2 -13766.508} C_VEL
LIN {X 0,Y 346.309,Z 853.114,A -85,B 0,C 180,E1 -13767.673,E2 -13767.673} C_VEL
LIN {X 0,Y 346.404,Z 853.871,A -85,B 0,C 180,E1 -13768.836,E2 -13768.836} C_VEL
LIN {X 0,Y 346.392,Z 854.194,A -85,B 0,C 180,E1 -13769.999,E2 -13769.999} C_VEL
LIN {X 0,Y 346.382,Z 854.112,A -85,B 0,C 180,E1 -13771.161,E2 -13771.161} C_VEL
LIN {X 0,Y 346.273,Z 853.616,A -85,B 0,C 180,E1 -13772.325,E2 -13772.325} C_VEL
LIN {X 0,Y 346.219,Z 852.669,A -85,B 0,C 180,E1 -13773.49,E2 -13773.49} C_VEL
LIN {X 0,Y 346.23,Z 851.304,A -85,B 0,C 180,E1 -13774.656,E2 -13774.656} C_VEL
LIN {X 0,Y 346.281,Z 848.443,A -85,B 0,C 180,E1 -13776.407,E2 -13776.407} C_VEL
LIN {X 0,Y 346.515,Z 844.529,A -85,B 0,C 180,E1 -13778.161,E2 -13778.161} C_VEL
LIN {X 0,Y 346.927,Z 839.469,A -85,B 0,C 180,E1 -13779.914,E2 -13779.914} C_VEL
LIN {X 0,Y 347.532,Z 833.115,A -85,B 0,C 180,E1 -13781.666,E2 -13781.666} C_VEL
LIN {X 0,Y 348.582,Z 825.275,A -85,B 0,C 180,E1 -13783.405,E2 -13783.405} C_VEL
LIN {X 0,Y 349.53,Z 817.287,A -85,B 0,C 180,E1 -13784.853,E2 -13784.853} C_VEL
LIN {X 0,Y 350.638,Z 807.576,A -85,B 0,C 180,E1 -13786.295,E2 -13786.295} C_VEL
LIN {X 0,Y 351.966,Z 796.868,A -85,B 0,C 180,E1 -13787.577,E2 -13787.577} C_VEL
LIN {X 0,Y 353.373,Z 784.971,A -85,B 0,C 180,E1 -13788.704,E2 -13788.704} C_VEL
LIN {X 0,Y 354.381,Z 774.609,A -85,B 0,C 180,E1 -13789.475,E2 -13789.475} C_VEL
LIN {X 0,Y 355.555,Z 760.799,A -85,B 0,C 180,E1 -13790.236,E2 -13790.236} C_VEL
LIN {X 0,Y 356.318,Z 747.854,A -85,B 0,C 180,E1 -13790.718,E2 -13790.718} C_VEL
LIN {X 0,Y 358.13,Z 679.747,A -85,B 0,C 180,E1 -13792.322,E2 -13792.322} C_VEL
LIN {X 0,Y 355.498,Z 659.534,A -85,B 0,C 180,E1 -13793.066,E2 -13793.066} C_VEL
LIN {X 0,Y 352.291,Z 641.786,A -85,B 0,C 180,E1 -13793.814,E2 -13793.814} C_VEL
LIN {X 0,Y 351.733,Z 638.898,A -85,B 0,C 180,E1 -13793.963,E2 -13793.963} C_VEL
LIN {X 0,Y 353.157,Z 627.151,A -85,B 0,C 180,E1 -13796.705,E2 -13796.705} C_VEL
LIN {X 0,Y 351.982,Z 619.852,A -85,B 0,C 180,E1 -13798.632,E2 -13798.632} C_VEL
LIN {X 0,Y 349.666,Z 609.797,A -85,B 0,C 180,E1 -13801.504,E2 -13801.504} C_VEL
LIN {X 0,Y 347.752,Z 602.169,A -85,B 0,C 180,E1 -13803.886,E2 -13803.886} C_VEL
LIN {X 0,Y 347.76,Z 602.168,A -85,B 0,C 180,E1 -13807.319,E2 -13807.319} C_VEL
LIN {X 0,Y 347.751,Z 602.173,A -85,B 0,C 180,E1 -13810.292,E2 -13810.292} C_VEL
LIN {X 0,Y 347.764,Z 602.169,A -85,B 0,C 180,E1 -13813.4,E2 -13813.4} C_VEL
LIN {X 0,Y 347.78,Z 602.164,A -85,B 0,C 180,E1 -13816.674,E2 -13816.674} C_VEL
LIN {X 0,Y 347.78,Z 602.167,A -85,B 0,C 180,E1 -13820.164,E2 -13820.164} C_VEL
LIN {X 0,Y 347.784,Z 602.161,A -85,B 0,C 180,E1 -13824.124,E2 -13824.124} C_VEL
LIN {X 0,Y 347.759,Z 602.162,A -85,B 0,C 180,E1 -13828.302,E2 -13828.302} C_VEL
LIN {X 0,Y 347.8,Z 602.154,A -85,B 0,C 180,E1 -13830.989,E2 -13830.989} C_VEL
LIN {X 0,Y 347.825,Z 602.153,A -85,B 0,C 180,E1 -13833.607,E2 -13833.607} C_VEL
LIN {X 0,Y 347.781,Z 602.161,A -85,B 0,C 180,E1 -13836.161,E2 -13836.161} C_VEL
LIN {X 0,Y 347.81,Z 602.155,A -85,B 0,C 180,E1 -13839.909,E2 -13839.909} C_VEL
LIN {X 0,Y 347.858,Z 602.151,A -85,B 0,C 180,E1 -13842.359,E2 -13842.359} C_VEL
LIN {X 0,Y 347.889,Z 602.148,A -85,B 0,C 180,E1 -13845.97,E2 -13845.97} C_VEL
LIN {X 0,Y 347.925,Z 602.145,A -85,B 0,C 180,E1 -13849.525,E2 -13849.525} C_VEL
LIN {X 0,Y 348.066,Z 602.13,A -85,B 0,C 180,E1 -13851.874,E2 -13851.874} C_VEL
LIN {X 0,Y 348.059,Z 602.13,A -85,B 0,C 180,E1 -13854.205,E2 -13854.205} C_VEL
LIN {X 0,Y 348.2,Z 602.112,A -85,B 0,C 180,E1 -13857.686,E2 -13857.686} C_VEL
LIN {X 0,Y 348.36,Z 602.094,A -85,B 0,C 180,E1 -13860,E2 -13860} C_VEL
LIN {X 0,Y 348.201,Z 602.113,A -85,B 0,C 180,E1 -13862.313,E2 -13862.313} C_VEL
LIN {X 0,Y 348.103,Z 602.128,A -85,B 0,C 180,E1 -13866.958,E2 -13866.958} C_VEL
LIN {X 0,Y 347.987,Z 602.207,A -85,B 0,C 180,E1 -13869.151,E2 -13869.151} C_VEL
LIN {X 0,Y 348.942,Z 606.88,A -85,B 0,C 180,E1 -13870.873,E2 -13870.873} C_VEL
LIN {X 0,Y 355.946,Z 622.243,A -85,B 0,C 180,E1 -13871.947,E2 -13871.947} C_VEL
LIN {X 0,Y 359.33,Z 630.671,A -85,B 0,C 180,E1 -13872.457,E2 -13872.457} C_VEL
LIN {X 0,Y 356.899,Z 712.361,A -85,B 0,C 180,E1 -13874.395,E2 -13874.395} C_VEL
LIN {X 0,Y 356.249,Z 725.952,A -85,B 0,C 180,E1 -13874.946,E2 -13874.946} C_VEL
LIN {X 0,Y 355.468,Z 738.171,A -85,B 0,C 180,E1 -13875.664,E2 -13875.664} C_VEL
LIN {X 0,Y 354.533,Z 749.538,A -85,B 0,C 180,E1 -13876.556,E2 -13876.556} C_VEL
LIN {X 0,Y 353.325,Z 761.469,A -85,B 0,C 180,E1 -13877.763,E2 -13877.763} C_VEL
LIN {X 0,Y 352.023,Z 771.875,A -85,B 0,C 180,E1 -13879.082,E2 -13879.082} C_VEL
LIN {X 0,Y 350.911,Z 780.575,A -85,B 0,C 180,E1 -13880.456,E2 -13880.456} C_VEL
LIN {X 0,Y 349.741,Z 788.982,A -85,B 0,C 180,E1 -13882.086,E2 -13882.086} C_VEL
LIN {X 0,Y 348.748,Z 795.979,A -85,B 0,C 180,E1 -13883.768,E2 -13883.768} C_VEL
LIN {X 0,Y 348.183,Z 800.433,A -85,B 0,C 180,E1 -13885.08,E2 -13885.08} C_VEL
LIN {X 0,Y 347.429,Z 805.975,A -85,B 0,C 180,E1 -13887.123,E2 -13887.123} C_VEL
LIN {X 0,Y 346.909,Z 809.88,A -85,B 0,C 180,E1 -13889.092,E2 -13889.092} C_VEL
LIN {X 0,Y 346.591,Z 811.794,A -85,B 0,C 180,E1 -13890.46,E2 -13890.46} C_VEL
LIN {X 0,Y 346.367,Z 813.173,A -85,B 0,C 180,E1 -13891.84,E2 -13891.84} C_VEL
LIN {X 0,Y 346.204,Z 814.07,A -85,B 0,C 180,E1 -13893.666,E2 -13893.666} C_VEL
LIN {X 0,Y 346.154,Z 813.868,A -85,B 0,C 180,E1 -13895.699,E2 -13895.699} C_VEL
LIN {X 0,Y 346.22,Z 812.496,A -85,B 0,C 180,E1 -13897.661,E2 -13897.661} C_VEL
LIN {X 0,Y 346.448,Z 810.018,A -85,B 0,C 180,E1 -13899.571,E2 -13899.571} C_VEL
LIN {X 0,Y 346.781,Z 806.47,A -85,B 0,C 180,E1 -13901.424,E2 -13901.424} C_VEL
LIN {X 0,Y 347.246,Z 801.094,A -85,B 0,C 180,E1 -13903.483,E2 -13903.483} C_VEL
LIN {X 0,Y 347.912,Z 794.436,A -85,B 0,C 180,E1 -13905.403,E2 -13905.403} C_VEL
LIN {X 0,Y 348.599,Z 787.577,A -85,B 0,C 180,E1 -13906.99,E2 -13906.99} C_VEL
LIN {X 0,Y 349.534,Z 778.661,A -85,B 0,C 180,E1 -13908.664,E2 -13908.664} C_VEL
LIN {X 0,Y 350.484,Z 769.251,A -85,B 0,C 180,E1 -13910.085,E2 -13910.085} C_VEL
LIN {X 0,Y 351.557,Z 757.634,A -85,B 0,C 180,E1 -13911.492,E2 -13911.492} C_VEL
LIN {X 0,Y 352.405,Z 746.644,A -85,B 0,C 180,E1 -13912.549,E2 -13912.549} C_VEL
LIN {X 0,Y 353.258,Z 734.833,A -85,B 0,C 180,E1 -13913.426,E2 -13913.426} C_VEL
LIN {X 0,Y 353.865,Z 721.305,A -85,B 0,C 180,E1 -13914.174,E2 -13914.174} C_VEL
LIN {X 0,Y 354.355,Z 708.513,A -85,B 0,C 180,E1 -13914.635,E2 -13914.635} C_VEL
LIN {X 0,Y 356.146,Z 627.855,A -85,B 0,C 180,E1 -13916.46,E2 -13916.46} C_VEL
LIN {X 0,Y 353.862,Z 620.158,A -85,B 0,C 180,E1 -13916.77,E2 -13916.77} C_VEL
LIN {X 0,Y 348.045,Z 603.52,A -85,B 0,C 180,E1 -13917.511,E2 -13917.511} C_VEL
LIN {X 0,Y 347.788,Z 602.166,A -85,B 0,C 180,E1 -13917.989,E2 -13917.989} C_VEL
LIN {X 0,Y 347.774,Z 602.161,A -85,B 0,C 180,E1 -13920.989,E2 -13920.989} C_VEL
LIN {X 0,Y 347.827,Z 602.156,A -85,B 0,C 180,E1 -13923.609,E2 -13923.609} C_VEL
LIN {X 0,Y 347.786,Z 602.165,A -85,B 0,C 180,E1 -13926.163,E2 -13926.163} C_VEL
LIN {X 0,Y 347.826,Z 602.158,A -85,B 0,C 180,E1 -13929.912,E2 -13929.912} C_VEL
LIN {X 0,Y 347.865,Z 602.155,A -85,B 0,C 180,E1 -13932.361,E2 -13932.361} C_VEL
LIN {X 0,Y 347.896,Z 602.149,A -85,B 0,C 180,E1 -13935.972,E2 -13935.972} C_VEL
LIN {X 0,Y 347.933,Z 602.141,A -85,B 0,C 180,E1 -13939.527,E2 -13939.527} C_VEL
LIN {X 0,Y 348.075,Z 602.125,A -85,B 0,C 180,E1 -13941.876,E2 -13941.876} C_VEL
LIN {X 0,Y 348.068,Z 602.128,A -85,B 0,C 180,E1 -13944.207,E2 -13944.207} C_VEL
LIN {X 0,Y 348.209,Z 602.107,A -85,B 0,C 180,E1 -13947.688,E2 -13947.688} C_VEL
LIN {X 0,Y 348.346,Z 602.091,A -85,B 0,C 180,E1 -13950.001,E2 -13950.001} C_VEL
LIN {X 0,Y 348.21,Z 602.11,A -85,B 0,C 180,E1 -13952.315,E2 -13952.315} C_VEL
LIN {X 0,Y 348.108,Z 602.123,A -85,B 0,C 180,E1 -13956.959,E2 -13956.959} C_VEL
LIN {X 0,Y 347.97,Z 602.138,A -85,B 0,C 180,E1 -13959.3,E2 -13959.3} C_VEL
LIN {X 0,Y 347.893,Z 602.152,A -85,B 0,C 180,E1 -13962.841,E2 -13962.841} C_VEL
LIN {X 0,Y 347.842,Z 602.155,A -85,B 0,C 180,E1 -13966.432,E2 -13966.432} C_VEL
LIN {X 0,Y 347.812,Z 602.157,A -85,B 0,C 180,E1 -13969.567,E2 -13969.567} C_VEL
LIN {X 0,Y 347.132,Z 602.245,A -85,B 0,C 180,E1 -13970.533,E2 -13970.533} C_VEL
LIN {X 0,Y 344.262,Z 602.599,A -85,B 0,C 180,E1 -13972.104,E2 -13972.104} C_VEL
LIN {X 0,Y 341.85,Z 602.901,A -85,B 0,C 180,E1 -13973.376,E2 -13973.376} C_VEL
LIN {X 0,Y 340.836,Z 603.027,A -85,B 0,C 180,E1 -13974.361,E2 -13974.361} C_VEL
LIN {X 0,Y 340.764,Z 603.037,A -85,B 0,C 180,E1 -13974.694,E2 -13974.694} C_VEL
LIN {X 0,Y 340.78,Z 603.034,A -85,B 0,C 180,E1 -13977.526,E2 -13977.526} C_VEL
LIN {X 0,Y 340.701,Z 603.048,A -85,B 0,C 180,E1 -13981.046,E2 -13981.046} C_VEL
LIN {X 0,Y 340.722,Z 603.045,A -85,B 0,C 180,E1 -13985.28,E2 -13985.28} C_VEL
LIN {X 0,Y 340.714,Z 603.041,A -85,B 0,C 180,E1 -13988.387,E2 -13988.387} C_VEL
LIN {X 0,Y 340.703,Z 603.042,A -85,B 0,C 180,E1 -13992.046,E2 -13992.046} C_VEL
LIN {X 0,Y 340.688,Z 603.049,A -85,B 0,C 180,E1 -13995.462,E2 -13995.462} C_VEL
LIN {X 0,Y 340.69,Z 603.044,A -85,B 0,C 180,E1 -13998.691,E2 -13998.691} C_VEL
LIN {X 0,Y 340.737,Z 603.041,A -85,B 0,C 180,E1 -14001.773,E2 -14001.773} C_VEL
LIN {X 0,Y 340.728,Z 603.045,A -85,B 0,C 180,E1 -14005.596,E2 -14005.596} C_VEL
LIN {X 0,Y 340.71,Z 603.042,A -85,B 0,C 180,E1 -14008.957,E2 -14008.957} C_VEL
LIN {X 0,Y 340.784,Z 603.032,A -85,B 0,C 180,E1 -14012.475,E2 -14012.475} C_VEL
LIN {X 0,Y 340.759,Z 603.04,A -85,B 0,C 180,E1 -14015.639,E2 -14015.639} C_VEL
LIN {X 0,Y 340.741,Z 603.04,A -85,B 0,C 180,E1 -14019.474,E2 -14019.474} C_VEL
LIN {X 0,Y 340.863,Z 603.027,A -85,B 0,C 180,E1 -14021.985,E2 -14021.985} C_VEL
LIN {X 0,Y 340.875,Z 603.024,A -85,B 0,C 180,E1 -14025.705,E2 -14025.705} C_VEL
LIN {X 0,Y 340.876,Z 603.021,A -85,B 0,C 180,E1 -14029.307,E2 -14029.307} C_VEL
LIN {X 0,Y 341.065,Z 602.997,A -85,B 0,C 180,E1 -14032.898,E2 -14032.898} C_VEL
LIN {X 0,Y 341.173,Z 602.985,A -85,B 0,C 180,E1 -14037.639,E2 -14037.639} C_VEL
LIN {X 0,Y 341.301,Z 602.972,A -85,B 0,C 180,E1 -14040,E2 -14040} C_VEL
LIN {X 0,Y 341.174,Z 602.988,A -85,B 0,C 180,E1 -14042.361,E2 -14042.361} C_VEL
LIN {X 0,Y 341.066,Z 602.997,A -85,B 0,C 180,E1 -14047.102,E2 -14047.102} C_VEL
LIN {X 0,Y 340.877,Z 603.023,A -85,B 0,C 180,E1 -14050.694,E2 -14050.694} C_VEL
LIN {X 0,Y 340.869,Z 603.026,A -85,B 0,C 180,E1 -14054.325,E2 -14054.325} C_VEL
LIN {X 0,Y 340.792,Z 603.036,A -85,B 0,C 180,E1 -14058.44,E2 -14058.44} C_VEL
LIN {X 0,Y 340.724,Z 603.04,A -85,B 0,C 180,E1 -14061.841,E2 -14061.841} C_VEL
LIN {X 0,Y 340.778,Z 603.032,A -85,B 0,C 180,E1 -14065.664,E2 -14065.664} C_VEL
LIN {X 0,Y 340.747,Z 603.039,A -85,B 0,C 180,E1 -14068.319,E2 -14068.319} C_VEL
LIN {X 0,Y 340.71,Z 603.044,A -85,B 0,C 180,E1 -14071.044,E2 -14071.044} C_VEL
LIN {X 0,Y 340.724,Z 603.041,A -85,B 0,C 180,E1 -14075.278,E2 -14075.278} C_VEL
LIN {X 0,Y 340.715,Z 603.042,A -85,B 0,C 180,E1 -14078.385,E2 -14078.385} C_VEL
LIN {X 0,Y 340.704,Z 603.042,A -85,B 0,C 180,E1 -14082.045,E2 -14082.045} C_VEL
LIN {X 0,Y 340.688,Z 603.046,A -85,B 0,C 180,E1 -14085.461,E2 -14085.461} C_VEL
LIN {X 0,Y 340.691,Z 603.046,A -85,B 0,C 180,E1 -14088.69,E2 -14088.69} C_VEL
LIN {X 0,Y 340.738,Z 603.038,A -85,B 0,C 180,E1 -14091.772,E2 -14091.772} C_VEL
LIN {X 0,Y 340.728,Z 603.043,A -85,B 0,C 180,E1 -14095.595,E2 -14095.595} C_VEL
LIN {X 0,Y 340.733,Z 603.212,A -85,B 0,C 180,E1 -14097.865,E2 -14097.865} C_VEL
LIN {X 0,Y 343.815,Z 617.279,A -85,B 0,C 180,E1 -14101.519,E2 -14101.519} C_VEL
LIN {X 0,Y 345.286,Z 625.58,A -85,B 0,C 180,E1 -14103.584,E2 -14103.584} C_VEL
LIN {X 0,Y 343.593,Z 641.542,A -85,B 0,C 180,E1 -14107.214,E2 -14107.214} C_VEL
LIN {X 0,Y 348.676,Z 680.603,A -85,B 0,C 180,E1 -14108.465,E2 -14108.465} C_VEL
LIN {X 0,Y 347.132,Z 750.456,A -85,B 0,C 180,E1 -14110.099,E2 -14110.099} C_VEL
LIN {X 0,Y 346.469,Z 763.938,A -85,B 0,C 180,E1 -14110.637,E2 -14110.637} C_VEL
LIN {X 0,Y 345.453,Z 776.825,A -85,B 0,C 180,E1 -14111.387,E2 -14111.387} C_VEL
LIN {X 0,Y 344.496,Z 788.665,A -85,B 0,C 180,E1 -14112.333,E2 -14112.333} C_VEL
LIN {X 0,Y 343.308,Z 800.098,A -85,B 0,C 180,E1 -14113.497,E2 -14113.497} C_VEL
LIN {X 0,Y 342.369,Z 809.955,A -85,B 0,C 180,E1 -14114.753,E2 -14114.753} C_VEL
LIN {X 0,Y 341.39,Z 819.769,A -85,B 0,C 180,E1 -14116.304,E2 -14116.304} C_VEL
LIN {X 0,Y 340.497,Z 828.831,A -85,B 0,C 180,E1 -14118.087,E2 -14118.087} C_VEL
LIN {X 0,Y 339.84,Z 836.087,A -85,B 0,C 180,E1 -14119.875,E2 -14119.875} C_VEL
LIN {X 0,Y 339.451,Z 841.848,A -85,B 0,C 180,E1 -14121.666,E2 -14121.666} C_VEL
LIN {X 0,Y 339.295,Z 846.361,A -85,B 0,C 180,E1 -14123.458,E2 -14123.458} C_VEL
LIN {X 0,Y 339.205,Z 849.733,A -85,B 0,C 180,E1 -14125.245,E2 -14125.245} C_VEL
LIN {X 0,Y 339.155,Z 851.389,A -85,B 0,C 180,E1 -14126.435,E2 -14126.435} C_VEL
LIN {X 0,Y 339.214,Z 852.627,A -85,B 0,C 180,E1 -14127.624,E2 -14127.624} C_VEL
LIN {X 0,Y 339.322,Z 853.424,A -85,B 0,C 180,E1 -14128.812,E2 -14128.812} C_VEL
LIN {X 0,Y 339.33,Z 853.767,A -85,B 0,C 180,E1 -14129.999,E2 -14129.999} C_VEL
LIN {X 0,Y 339.3,Z 853.699,A -85,B 0,C 180,E1 -14131.186,E2 -14131.186} C_VEL
LIN {X 0,Y 339.176,Z 853.221,A -85,B 0,C 180,E1 -14132.374,E2 -14132.374} C_VEL
LIN {X 0,Y 339.139,Z 852.307,A -85,B 0,C 180,E1 -14133.563,E2 -14133.563} C_VEL
LIN {X 0,Y 339.126,Z 850.954,A -85,B 0,C 180,E1 -14134.754,E2 -14134.754} C_VEL
LIN {X 0,Y 339.202,Z 848.122,A -85,B 0,C 180,E1 -14136.542,E2 -14136.542} C_VEL
LIN {X 0,Y 339.452,Z 844.245,A -85,B 0,C 180,E1 -14138.332,E2 -14138.332} C_VEL
LIN {X 0,Y 339.905,Z 839.236,A -85,B 0,C 180,E1 -14140.121,E2 -14140.121} C_VEL
LIN {X 0,Y 340.553,Z 832.947,A -85,B 0,C 180,E1 -14141.908,E2 -14141.908} C_VEL
LIN {X 0,Y 341.649,Z 825.161,A -85,B 0,C 180,E1 -14143.682,E2 -14143.682} C_VEL
LIN {X 0,Y 342.647,Z 817.295,A -85,B 0,C 180,E1 -14145.149,E2 -14145.149} C_VEL
LIN {X 0,Y 343.819,Z 807.624,A -85,B 0,C 180,E1 -14146.628,E2 -14146.628} C_VEL
LIN {X 0,Y 345.371,Z 795.703,A -85,B 0,C 180,E1 -14148.077,E2 -14148.077} C_VEL
LIN {X 0,Y 346.858,Z 783.567,A -85,B 0,C 180,E1 -14149.222,E2 -14149.222} C_VEL
LIN {X 0,Y 347.924,Z 773.016,A -85,B 0,C 180,E1 -14150.005,E2 -14150.005} C_VEL
LIN {X 0,Y 349.122,Z 759.659,A -85,B 0,C 180,E1 -14150.741,E2 -14150.741} C_VEL
LIN {X 0,Y 349.859,Z 746.499,A -85,B 0,C 180,E1 -14151.23,E2 -14151.23} C_VEL
LIN {X 0,Y 351.723,Z 680.119,A -85,B 0,C 180,E1 -14152.831,E2 -14152.831} C_VEL
LIN {X 0,Y 349.108,Z 660.08,A -85,B 0,C 180,E1 -14153.592,E2 -14153.592} C_VEL
LIN {X 0,Y 345.631,Z 641.184,A -85,B 0,C 180,E1 -14154.435,E2 -14154.435} C_VEL
LIN {X 0,Y 345.087,Z 638.341,A -85,B 0,C 180,E1 -14154.6,E2 -14154.6} C_VEL
LIN {X 0,Y 346.292,Z 629.336,A -85,B 0,C 180,E1 -14156.749,E2 -14156.749} C_VEL
LIN {X 0,Y 345.841,Z 625.097,A -85,B 0,C 180,E1 -14157.864,E2 -14157.864} C_VEL
LIN {X 0,Y 343.663,Z 614.799,A -85,B 0,C 180,E1 -14160.805,E2 -14160.805} C_VEL
LIN {X 0,Y 341.255,Z 605.225,A -85,B 0,C 180,E1 -14163.782,E2 -14163.782} C_VEL
LIN {X 0,Y 340.709,Z 603.047,A -85,B 0,C 180,E1 -14164.539,E2 -14164.539} C_VEL
LIN {X 0,Y 340.714,Z 603.049,A -85,B 0,C 180,E1 -14168.387,E2 -14168.387} C_VEL
LIN {X 0,Y 340.729,Z 603.048,A -85,B 0,C 180,E1 -14172.051,E2 -14172.051} C_VEL
LIN {X 0,Y 340.746,Z 603.042,A -85,B 0,C 180,E1 -14175.471,E2 -14175.471} C_VEL
LIN {X 0,Y 340.72,Z 603.042,A -85,B 0,C 180,E1 -14178.695,E2 -14178.695} C_VEL
LIN {X 0,Y 340.735,Z 603.04,A -85,B 0,C 180,E1 -14181.773,E2 -14181.773} C_VEL
LIN {X 0,Y 340.716,Z 603.041,A -85,B 0,C 180,E1 -14185.594,E2 -14185.594} C_VEL
LIN {X 0,Y 340.711,Z 603.04,A -85,B 0,C 180,E1 -14188.956,E2 -14188.956} C_VEL
LIN {X 0,Y 340.773,Z 603.036,A -85,B 0,C 180,E1 -14192.473,E2 -14192.473} C_VEL
LIN {X 0,Y 340.749,Z 603.038,A -85,B 0,C 180,E1 -14195.638,E2 -14195.638} C_VEL
LIN {X 0,Y 340.741,Z 603.036,A -85,B 0,C 180,E1 -14199.474,E2 -14199.474} C_VEL
LIN {X 0,Y 340.85,Z 603.026,A -85,B 0,C 180,E1 -14201.984,E2 -14201.984} C_VEL
LIN {X 0,Y 340.861,Z 603.022,A -85,B 0,C 180,E1 -14205.704,E2 -14205.704} C_VEL
LIN {X 0,Y 340.867,Z 603.024,A -85,B 0,C 180,E1 -14209.306,E2 -14209.306} C_VEL
LIN {X 0,Y 341.067,Z 602.999,A -85,B 0,C 180,E1 -14212.898,E2 -14212.898} C_VEL
LIN {X 0,Y 341.162,Z 602.988,A -85,B 0,C 180,E1 -14217.639,E2 -14217.639} C_VEL
LIN {X 0,Y 341.309,Z 602.972,A -85,B 0,C 180,E1 -14220,E2 -14220} C_VEL
LIN {X 0,Y 341.163,Z 602.989,A -85,B 0,C 180,E1 -14222.361,E2 -14222.361} C_VEL
LIN {X 0,Y 341.071,Z 603.003,A -85,B 0,C 180,E1 -14227.102,E2 -14227.102} C_VEL
LIN {X 0,Y 341.028,Z 603.175,A -85,B 0,C 180,E1 -14228.562,E2 -14228.562} C_VEL
LIN {X 0,Y 341.911,Z 607.46,A -85,B 0,C 180,E1 -14230.196,E2 -14230.196} C_VEL
LIN {X 0,Y 349.227,Z 623.178,A -85,B 0,C 180,E1 -14231.367,E2 -14231.367} C_VEL
LIN {X 0,Y 352.975,Z 632.268,A -85,B 0,C 180,E1 -14231.958,E2 -14231.958} C_VEL
LIN {X 0,Y 350.481,Z 713.089,A -85,B 0,C 180,E1 -14233.924,E2 -14233.924} C_VEL
LIN {X 0,Y 349.798,Z 726.445,A -85,B 0,C 180,E1 -14234.476,E2 -14234.476} C_VEL
LIN {X 0,Y 348.922,Z 739.305,A -85,B 0,C 180,E1 -14235.254,E2 -14235.254} C_VEL
LIN {X 0,Y 347.99,Z 750.035,A -85,B 0,C 180,E1 -14236.123,E2 -14236.123} C_VEL
LIN {X 0,Y 346.815,Z 760.9,A -85,B 0,C 180,E1 -14237.232,E2 -14237.232} C_VEL
LIN {X 0,Y 345.505,Z 771.146,A -85,B 0,C 180,E1 -14238.532,E2 -14238.532} C_VEL
LIN {X 0,Y 344.184,Z 780.902,A -85,B 0,C 180,E1 -14240.072,E2 -14240.072} C_VEL
LIN {X 0,Y 342.856,Z 789.932,A -85,B 0,C 180,E1 -14241.864,E2 -14241.864} C_VEL
LIN {X 0,Y 341.781,Z 797.066,A -85,B 0,C 180,E1 -14243.639,E2 -14243.639} C_VEL
LIN {X 0,Y 340.93,Z 803.325,A -85,B 0,C 180,E1 -14245.652,E2 -14245.652} C_VEL
LIN {X 0,Y 340.302,Z 807.479,A -85,B 0,C 180,E1 -14247.375,E2 -14247.375} C_VEL
LIN {X 0,Y 339.699,Z 811.449,A -85,B 0,C 180,E1 -14249.668,E2 -14249.668} C_VEL
LIN {X 0,Y 339.284,Z 813.707,A -85,B 0,C 180,E1 -14251.869,E2 -14251.869} C_VEL
LIN {X 0,Y 339.1,Z 814.536,A -85,B 0,C 180,E1 -14254.027,E2 -14254.027} C_VEL
LIN {X 0,Y 339.076,Z 814.092,A -85,B 0,C 180,E1 -14256.068,E2 -14256.068} C_VEL
LIN {X 0,Y 339.203,Z 812.061,A -85,B 0,C 180,E1 -14258.431,E2 -14258.431} C_VEL
LIN {X 0,Y 339.574,Z 808.522,A -85,B 0,C 180,E1 -14260.687,E2 -14260.687} C_VEL
LIN {X 0,Y 339.879,Z 804.727,A -85,B 0,C 180,E1 -14262.398,E2 -14262.398} C_VEL
LIN {X 0,Y 340.344,Z 799.913,A -85,B 0,C 180,E1 -14264.09,E2 -14264.09} C_VEL
LIN {X 0,Y 340.978,Z 793.94,A -85,B 0,C 180,E1 -14265.774,E2 -14265.774} C_VEL
LIN {X 0,Y 341.719,Z 786.625,A -85,B 0,C 180,E1 -14267.448,E2 -14267.448} C_VEL
LIN {X 0,Y 342.732,Z 777.59,A -85,B 0,C 180,E1 -14269.108,E2 -14269.108} C_VEL
LIN {X 0,Y 343.744,Z 767.59,A -85,B 0,C 180,E1 -14270.592,E2 -14270.592} C_VEL
LIN {X 0,Y 344.715,Z 757.321,A -85,B 0,C 180,E1 -14271.827,E2 -14271.827} C_VEL
LIN {X 0,Y 345.651,Z 745.578,A -85,B 0,C 180,E1 -14272.945,E2 -14272.945} C_VEL
LIN {X 0,Y 346.537,Z 732.56,A -85,B 0,C 180,E1 -14273.893,E2 -14273.893} C_VEL
LIN {X 0,Y 347.112,Z 719.921,A -85,B 0,C 180,E1 -14274.559,E2 -14274.559} C_VEL
LIN {X 0,Y 347.633,Z 706.299,A -85,B 0,C 180,E1 -14275.019,E2 -14275.019} C_VEL
LIN {X 0,Y 349.332,Z 628.556,A -85,B 0,C 180,E1 -14276.814,E2 -14276.814} C_VEL
LIN {X 0,Y 342.459,Z 608.45,A -85,B 0,C 180,E1 -14277.711,E2 -14277.711} C_VEL
LIN {X 0,Y 340.878,Z 603.772,A -85,B 0,C 180,E1 -14277.96,E2 -14277.96} C_VEL
LIN {X 0,Y 340.749,Z 603.04,A -85,B 0,C 180,E1 -14278.27,E2 -14278.27} C_VEL
LIN {X 0,Y 340.724,Z 603.042,A -85,B 0,C 180,E1 -14281.681,E2 -14281.681} C_VEL
LIN {X 0,Y 340.769,Z 603.037,A -85,B 0,C 180,E1 -14284.337,E2 -14284.337} C_VEL
LIN {X 0,Y 340.74,Z 603.043,A -85,B 0,C 180,E1 -14288.208,E2 -14288.208} C_VEL
LIN {X 0,Y 340.857,Z 603.027,A -85,B 0,C 180,E1 -14291.986,E2 -14291.986} C_VEL
LIN {X 0,Y 340.868,Z 603.022,A -85,B 0,C 180,E1 -14295.706,E2 -14295.706} C_VEL
LIN {X 0,Y 340.875,Z 603.02,A -85,B 0,C 180,E1 -14299.308,E2 -14299.308} C_VEL
LIN {X 0,Y 341.076,Z 602.997,A -85,B 0,C 180,E1 -14302.9,E2 -14302.9} C_VEL
LIN {X 0,Y 341.171,Z 602.984,A -85,B 0,C 180,E1 -14307.64,E2 -14307.64} C_VEL
LIN {X 0,Y 341.296,Z 602.969,A -85,B 0,C 180,E1 -14310.001,E2 -14310.001} C_VEL
LIN {X 0,Y 341.172,Z 602.987,A -85,B 0,C 180,E1 -14312.362,E2 -14312.362} C_VEL
LIN {X 0,Y 341.078,Z 602.997,A -85,B 0,C 180,E1 -14317.103,E2 -14317.103} C_VEL
LIN {X 0,Y 340.873,Z 603.027,A -85,B 0,C 180,E1 -14320.695,E2 -14320.695} C_VEL
LIN {X 0,Y 340.865,Z 603.023,A -85,B 0,C 180,E1 -14324.326,E2 -14324.326} C_VEL
LIN {X 0,Y 340.84,Z 603.027,A -85,B 0,C 180,E1 -14328.467,E2 -14328.467} C_VEL
LIN {X 0,Y 340.757,Z 603.035,A -85,B 0,C 180,E1 -14331.858,E2 -14331.858} C_VEL
LIN {X 0,Y 340.764,Z 603.037,A -85,B 0,C 180,E1 -14334.694,E2 -14334.694} C_VEL
LIN {X 0,Y 340.114,Z 603.124,A -85,B 0,C 180,E1 -14335.681,E2 -14335.681} C_VEL
LIN {X 0,Y 337.229,Z 603.483,A -85,B 0,C 180,E1 -14337.285,E2 -14337.285} C_VEL
LIN {X 0,Y 334.782,Z 603.782,A -85,B 0,C 180,E1 -14338.584,E2 -14338.584} C_VEL
LIN {X 0,Y 333.752,Z 603.909,A -85,B 0,C 180,E1 -14339.591,E2 -14339.591} C_VEL
LIN {X 0,Y 333.679,Z 603.916,A -85,B 0,C 180,E1 -14339.932,E2 -14339.932} C_VEL
LIN {X 0,Y 333.64,Z 603.927,A -85,B 0,C 180,E1 -14343.209,E2 -14343.209} C_VEL
LIN {X 0,Y 333.68,Z 603.917,A -85,B 0,C 180,E1 -14346.14,E2 -14346.14} C_VEL
LIN {X 0,Y 333.65,Z 603.926,A -85,B 0,C 180,E1 -14349.193,E2 -14349.193} C_VEL
LIN {X 0,Y 333.637,Z 603.922,A -85,B 0,C 180,E1 -14352.501,E2 -14352.501} C_VEL
LIN {X 0,Y 333.626,Z 603.924,A -85,B 0,C 180,E1 -14355.96,E2 -14355.96} C_VEL
LIN {X 0,Y 333.652,Z 603.925,A -85,B 0,C 180,E1 -14359.316,E2 -14359.316} C_VEL
LIN {X 0,Y 333.669,Z 603.921,A -85,B 0,C 180,E1 -14363.169,E2 -14363.169} C_VEL
LIN {X 0,Y 333.644,Z 603.921,A -85,B 0,C 180,E1 -14366.793,E2 -14366.793} C_VEL
LIN {X 0,Y 333.708,Z 603.919,A -85,B 0,C 180,E1 -14369.711,E2 -14369.711} C_VEL
LIN {X 0,Y 333.748,Z 603.909,A -85,B 0,C 180,E1 -14372.402,E2 -14372.402} C_VEL
LIN {X 0,Y 333.731,Z 603.911,A -85,B 0,C 180,E1 -14375.091,E2 -14375.091} C_VEL
LIN {X 0,Y 333.679,Z 603.917,A -85,B 0,C 180,E1 -14379.019,E2 -14379.019} C_VEL
LIN {X 0,Y 333.8,Z 603.905,A -85,B 0,C 180,E1 -14381.59,E2 -14381.59} C_VEL
LIN {X 0,Y 333.814,Z 603.903,A -85,B 0,C 180,E1 -14385.577,E2 -14385.577} C_VEL
LIN {X 0,Y 333.839,Z 603.897,A -85,B 0,C 180,E1 -14389.078,E2 -14389.078} C_VEL
LIN {X 0,Y 334.012,Z 603.876,A -85,B 0,C 180,E1 -14392.747,E2 -14392.747} C_VEL
LIN {X 0,Y 333.813,Z 603.9,A -85,B 0,C 180,E1 -14395.169,E2 -14395.169} C_VEL
LIN {X 0,Y 334.111,Z 603.864,A -85,B 0,C 180,E1 -14397.589,E2 -14397.589} C_VEL
LIN {X 0,Y 334.252,Z 603.85,A -85,B 0,C 180,E1 -14400,E2 -14400} C_VEL
LIN {X 0,Y 334.111,Z 603.867,A -85,B 0,C 180,E1 -14402.411,E2 -14402.411} C_VEL
LIN {X 0,Y 334.021,Z 603.878,A -85,B 0,C 180,E1 -14406.039,E2 -14406.039} C_VEL
LIN {X 0,Y 333.965,Z 603.886,A -85,B 0,C 180,E1 -14408.471,E2 -14408.471} C_VEL
LIN {X 0,Y 333.797,Z 603.906,A -85,B 0,C 180,E1 -14412.155,E2 -14412.155} C_VEL
LIN {X 0,Y 333.814,Z 603.904,A -85,B 0,C 180,E1 -14414.634,E2 -14414.634} C_VEL
LIN {X 0,Y 333.729,Z 603.916,A -85,B 0,C 180,E1 -14418.618,E2 -14418.618} C_VEL
LIN {X 0,Y 333.663,Z 603.922,A -85,B 0,C 180,E1 -14422.28,E2 -14422.28} C_VEL
LIN {X 0,Y 333.742,Z 603.911,A -85,B 0,C 180,E1 -14426.246,E2 -14426.246} C_VEL
LIN {X 0,Y 333.717,Z 603.916,A -85,B 0,C 180,E1 -14428.972,E2 -14428.972} C_VEL
LIN {X 0,Y 333.649,Z 603.925,A -85,B 0,C 180,E1 -14432.587,E2 -14432.587} C_VEL
LIN {X 0,Y 333.682,Z 603.917,A -85,B 0,C 180,E1 -14436.139,E2 -14436.139} C_VEL
LIN {X 0,Y 333.652,Z 603.923,A -85,B 0,C 180,E1 -14439.192,E2 -14439.192} C_VEL
LIN {X 0,Y 333.638,Z 603.924,A -85,B 0,C 180,E1 -14442.5,E2 -14442.5} C_VEL
LIN {X 0,Y 333.626,Z 603.923,A -85,B 0,C 180,E1 -14445.958,E2 -14445.958} C_VEL
LIN {X 0,Y 333.653,Z 603.924,A -85,B 0,C 180,E1 -14449.315,E2 -14449.315} C_VEL
LIN {X 0,Y 333.67,Z 603.924,A -85,B 0,C 180,E1 -14453.167,E2 -14453.167} C_VEL
LIN {X 0,Y 333.642,Z 603.926,A -85,B 0,C 180,E1 -14456.791,E2 -14456.791} C_VEL
LIN {X 0,Y 333.686,Z 604.044,A -85,B 0,C 180,E1 -14457.525,E2 -14457.525} C_VEL
LIN {X 0,Y 336.81,Z 618.324,A -85,B 0,C 180,E1 -14461.318,E2 -14461.318} C_VEL
LIN {X 0,Y 338.279,Z 626.088,A -85,B 0,C 180,E1 -14463.299,E2 -14463.299} C_VEL
LIN {X 0,Y 337.233,Z 636.37,A -85,B 0,C 180,E1 -14465.694,E2 -14465.694} C_VEL
LIN {X 0,Y 336.696,Z 641.189,A -85,B 0,C 180,E1 -14466.81,E2 -14466.81} C_VEL
LIN {X 0,Y 341.896,Z 681.362,A -85,B 0,C 180,E1 -14468.126,E2 -14468.126} C_VEL
LIN {X 0,Y 340.273,Z 750.896,A -85,B 0,C 180,E1 -14469.798,E2 -14469.798} C_VEL
LIN {X 0,Y 339.517,Z 764.825,A -85,B 0,C 180,E1 -14470.382,E2 -14470.382} C_VEL
LIN {X 0,Y 338.609,Z 776.294,A -85,B 0,C 180,E1 -14471.075,E2 -14471.075} C_VEL
LIN {X 0,Y 337.533,Z 788.956,A -85,B 0,C 180,E1 -14472.113,E2 -14472.113} C_VEL
LIN {X 0,Y 336.32,Z 800.266,A -85,B 0,C 180,E1 -14473.301,E2 -14473.301} C_VEL
LIN {X 0,Y 335.367,Z 809.98,A -85,B 0,C 180,E1 -14474.577,E2 -14474.577} C_VEL
LIN {X 0,Y 334.464,Z 818.907,A -85,B 0,C 180,E1 -14476.015,E2 -14476.015} C_VEL
LIN {X 0,Y 333.526,Z 828.049,A -85,B 0,C 180,E1 -14477.834,E2 -14477.834} C_VEL
LIN {X 0,Y 332.81,Z 835.391,A -85,B 0,C 180,E1 -14479.658,E2 -14479.658} C_VEL
LIN {X 0,Y 332.401,Z 841.221,A -85,B 0,C 180,E1 -14481.488,E2 -14481.488} C_VEL
LIN {X 0,Y 332.216,Z 845.783,A -85,B 0,C 180,E1 -14483.317,E2 -14483.317} C_VEL
LIN {X 0,Y 332.121,Z 849.204,A -85,B 0,C 180,E1 -14485.143,E2 -14485.143} C_VEL
LIN {X 0,Y 332.08,Z 850.882,A -85,B 0,C 180,E1 -14486.359,E2 -14486.359} C_VEL
LIN {X 0,Y 332.12,Z 852.14,A -85,B 0,C 180,E1 -14487.573,E2 -14487.573} C_VEL
LIN {X 0,Y 332.242,Z 852.974,A -85,B 0,C 180,E1 -14488.787,E2 -14488.787} C_VEL
LIN {X 0,Y 332.27,Z 853.339,A -85,B 0,C 180,E1 -14489.999,E2 -14489.999} C_VEL
LIN {X 0,Y 332.205,Z 853.286,A -85,B 0,C 180,E1 -14491.211,E2 -14491.211} C_VEL
LIN {X 0,Y 332.081,Z 852.825,A -85,B 0,C 180,E1 -14492.425,E2 -14492.425} C_VEL
LIN {X 0,Y 332.06,Z 851.947,A -85,B 0,C 180,E1 -14493.639,E2 -14493.639} C_VEL
LIN {X 0,Y 332.074,Z 849.145,A -85,B 0,C 180,E1 -14495.896,E2 -14495.896} C_VEL
LIN {X 0,Y 332.304,Z 845.389,A -85,B 0,C 180,E1 -14497.9,E2 -14497.9} C_VEL
LIN {X 0,Y 332.702,Z 840.815,A -85,B 0,C 180,E1 -14499.728,E2 -14499.728} C_VEL
LIN {X 0,Y 333.29,Z 835.023,A -85,B 0,C 180,E1 -14501.554,E2 -14501.554} C_VEL
LIN {X 0,Y 334.332,Z 827.833,A -85,B 0,C 180,E1 -14503.368,E2 -14503.368} C_VEL
LIN {X 0,Y 335.486,Z 819.257,A -85,B 0,C 180,E1 -14505.105,E2 -14505.105} C_VEL
LIN {X 0,Y 336.869,Z 808.753,A -85,B 0,C 180,E1 -14506.825,E2 -14506.825} C_VEL
LIN {X 0,Y 338.29,Z 798.555,A -85,B 0,C 180,E1 -14508.156,E2 -14508.156} C_VEL
LIN {X 0,Y 339.831,Z 787.315,A -85,B 0,C 180,E1 -14509.322,E2 -14509.322} C_VEL
LIN {X 0,Y 340.96,Z 776.819,A -85,B 0,C 180,E1 -14510.196,E2 -14510.196} C_VEL
LIN {X 0,Y 342.253,Z 764.407,A -85,B 0,C 180,E1 -14510.98,E2 -14510.98} C_VEL
LIN {X 0,Y 343.184,Z 751.721,A -85,B 0,C 180,E1 -14511.55,E2 -14511.55} C_VEL
LIN {X 0,Y 343.831,Z 734.614,A -85,B 0,C 180,E1 -14512.025,E2 -14512.025} C_VEL
LIN {X 0,Y 345.391,Z 680.881,A -85,B 0,C 180,E1 -14513.347,E2 -14513.347} C_VEL
LIN {X 0,Y 342.768,Z 660.454,A -85,B 0,C 180,E1 -14514.16,E2 -14514.16} C_VEL
LIN {X 0,Y 339.093,Z 640.841,A -85,B 0,C 180,E1 -14515.077,E2 -14515.077} C_VEL
LIN {X 0,Y 338.472,Z 637.846,A -85,B 0,C 180,E1 -14515.257,E2 -14515.257} C_VEL
LIN {X 0,Y 339.476,Z 630.326,A -85,B 0,C 180,E1 -14517.1,E2 -14517.1} C_VEL
LIN {X 0,Y 338.234,Z 622.762,A -85,B 0,C 180,E1 -14519.226,E2 -14519.226} C_VEL
LIN {X 0,Y 335.993,Z 612.85,A -85,B 0,C 180,E1 -14522.233,E2 -14522.233} C_VEL
LIN {X 0,Y 333.667,Z 603.923,A -85,B 0,C 180,E1 -14525.212,E2 -14525.212} C_VEL
LIN {X 0,Y 333.668,Z 603.924,A -85,B 0,C 180,E1 -14529.187,E2 -14529.187} C_VEL
LIN {X 0,Y 333.671,Z 603.924,A -85,B 0,C 180,E1 -14532.507,E2 -14532.507} C_VEL
LIN {X 0,Y 333.687,Z 603.923,A -85,B 0,C 180,E1 -14535.97,E2 -14535.97} C_VEL
LIN {X 0,Y 333.696,Z 603.918,A -85,B 0,C 180,E1 -14539.303,E2 -14539.303} C_VEL
LIN {X 0,Y 333.661,Z 603.918,A -85,B 0,C 180,E1 -14543.166,E2 -14543.166} C_VEL
LIN {X 0,Y 333.635,Z 603.925,A -85,B 0,C 180,E1 -14546.791,E2 -14546.791} C_VEL
LIN {X 0,Y 333.698,Z 603.914,A -85,B 0,C 180,E1 -14549.709,E2 -14549.709} C_VEL
LIN {X 0,Y 333.738,Z 603.911,A -85,B 0,C 180,E1 -14552.4,E2 -14552.4} C_VEL
LIN {X 0,Y 333.72,Z 603.914,A -85,B 0,C 180,E1 -14555.09,E2 -14555.09} C_VEL
LIN {X 0,Y 333.674,Z 603.917,A -85,B 0,C 180,E1 -14559.019,E2 -14559.019} C_VEL
LIN {X 0,Y 333.786,Z 603.907,A -85,B 0,C 180,E1 -14561.589,E2 -14561.589} C_VEL
LIN {X 0,Y 333.8,Z 603.901,A -85,B 0,C 180,E1 -14565.576,E2 -14565.576} C_VEL
LIN {X 0,Y 333.829,Z 603.902,A -85,B 0,C 180,E1 -14569.078,E2 -14569.078} C_VEL
LIN {X 0,Y 334.017,Z 603.876,A -85,B 0,C 180,E1 -14572.747,E2 -14572.747} C_VEL
LIN {X 0,Y 333.805,Z 603.904,A -85,B 0,C 180,E1 -14575.169,E2 -14575.169} C_VEL
LIN {X 0,Y 334.099,Z 603.868,A -85,B 0,C 180,E1 -14577.589,E2 -14577.589} C_VEL
LIN {X 0,Y 334.259,Z 603.85,A -85,B 0,C 180,E1 -14580,E2 -14580} C_VEL
LIN {X 0,Y 334.124,Z 603.866,A -85,B 0,C 180,E1 -14582.411,E2 -14582.411} C_VEL
LIN {X 0,Y 334.02,Z 603.881,A -85,B 0,C 180,E1 -14587.252,E2 -14587.252} C_VEL
LIN {X 0,Y 334.005,Z 603.956,A -85,B 0,C 180,E1 -14587.861,E2 -14587.861} C_VEL
LIN {X 0,Y 334.881,Z 608.14,A -85,B 0,C 180,E1 -14589.481,E2 -14589.481} C_VEL
LIN {X 0,Y 343.114,Z 625.368,A -85,B 0,C 180,E1 -14590.847,E2 -14590.847} C_VEL
LIN {X 0,Y 346.686,Z 634.16,A -85,B 0,C 180,E1 -14591.437,E2 -14591.437} C_VEL
LIN {X 0,Y 344.081,Z 713.84,A -85,B 0,C 180,E1 -14593.435,E2 -14593.435} C_VEL
LIN {X 0,Y 343.364,Z 727.008,A -85,B 0,C 180,E1 -14593.991,E2 -14593.991} C_VEL
LIN {X 0,Y 342.427,Z 740.01,A -85,B 0,C 180,E1 -14594.796,E2 -14594.796} C_VEL
LIN {X 0,Y 341.275,Z 752.315,A -85,B 0,C 180,E1 -14595.835,E2 -14595.835} C_VEL
LIN {X 0,Y 339.98,Z 763.638,A -85,B 0,C 180,E1 -14597.057,E2 -14597.057} C_VEL
LIN {X 0,Y 338.5,Z 773.956,A -85,B 0,C 180,E1 -14598.459,E2 -14598.459} C_VEL
LIN {X 0,Y 337.111,Z 783.456,A -85,B 0,C 180,E1 -14600.073,E2 -14600.073} C_VEL
LIN {X 0,Y 335.85,Z 791.648,A -85,B 0,C 180,E1 -14601.804,E2 -14601.804} C_VEL
LIN {X 0,Y 334.588,Z 799.256,A -85,B 0,C 180,E1 -14603.85,E2 -14603.85} C_VEL
LIN {X 0,Y 333.852,Z 804.558,A -85,B 0,C 180,E1 -14605.679,E2 -14605.679} C_VEL
LIN {X 0,Y 333.164,Z 808.954,A -85,B 0,C 180,E1 -14607.651,E2 -14607.651} C_VEL
LIN {X 0,Y 332.565,Z 812.477,A -85,B 0,C 180,E1 -14609.956,E2 -14609.956} C_VEL
LIN {X 0,Y 332.167,Z 814.427,A -85,B 0,C 180,E1 -14612.189,E2 -14612.189} C_VEL
LIN {X 0,Y 332.011,Z 814.994,A -85,B 0,C 180,E1 -14614.359,E2 -14614.359} C_VEL
LIN {X 0,Y 331.994,Z 814.278,A -85,B 0,C 180,E1 -14616.448,E2 -14616.448} C_VEL
LIN {X 0,Y 332.117,Z 812.419,A -85,B 0,C 180,E1 -14618.47,E2 -14618.47} C_VEL
LIN {X 0,Y 332.463,Z 809.443,A -85,B 0,C 180,E1 -14620.449,E2 -14620.449} C_VEL
LIN {X 0,Y 332.836,Z 805.052,A -85,B 0,C 180,E1 -14622.508,E2 -14622.508} C_VEL
LIN {X 0,Y 333.397,Z 799.367,A -85,B 0,C 180,E1 -14624.509,E2 -14624.509} C_VEL
LIN {X 0,Y 334.085,Z 792.921,A -85,B 0,C 180,E1 -14626.282,E2 -14626.282} C_VEL
LIN {X 0,Y 334.934,Z 785.062,A -85,B 0,C 180,E1 -14628.023,E2 -14628.023} C_VEL
LIN {X 0,Y 335.998,Z 775.598,A -85,B 0,C 180,E1 -14629.716,E2 -14629.716} C_VEL
LIN {X 0,Y 337.067,Z 765.229,A -85,B 0,C 180,E1 -14631.198,E2 -14631.198} C_VEL
LIN {X 0,Y 338.041,Z 754.647,A -85,B 0,C 180,E1 -14632.416,E2 -14632.416} C_VEL
LIN {X 0,Y 339.056,Z 742.832,A -85,B 0,C 180,E1 -14633.495,E2 -14633.495} C_VEL
LIN {X 0,Y 339.887,Z 729.64,A -85,B 0,C 180,E1 -14634.398,E2 -14634.398} C_VEL
LIN {X 0,Y 340.481,Z 716.445,A -85,B 0,C 180,E1 -14635.041,E2 -14635.041} C_VEL
LIN {X 0,Y 340.93,Z 702.288,A -85,B 0,C 180,E1 -14635.459,E2 -14635.459} C_VEL
LIN {X 0,Y 342.635,Z 629.782,A -85,B 0,C 180,E1 -14637.163,E2 -14637.163} C_VEL
LIN {X 0,Y 333.752,Z 604.22,A -85,B 0,C 180,E1 -14638.37,E2 -14638.37} C_VEL
LIN {X 0,Y 333.687,Z 603.918,A -85,B 0,C 180,E1 -14638.584,E2 -14638.584} C_VEL
LIN {X 0,Y 333.736,Z 603.912,A -85,B 0,C 180,E1 -14642.402,E2 -14642.402} C_VEL
LIN {X 0,Y 333.724,Z 603.911,A -85,B 0,C 180,E1 -14645.092,E2 -14645.092} C_VEL
LIN {X 0,Y 333.691,Z 603.915,A -85,B 0,C 180,E1 -14649.021,E2 -14649.021} C_VEL
LIN {X 0,Y 333.793,Z 603.904,A -85,B 0,C 180,E1 -14651.591,E2 -14651.591} C_VEL
LIN {X 0,Y 333.807,Z 603.901,A -85,B 0,C 180,E1 -14655.578,E2 -14655.578} C_VEL
LIN {X 0,Y 333.837,Z 603.898,A -85,B 0,C 180,E1 -14659.08,E2 -14659.08} C_VEL
LIN {X 0,Y 334.026,Z 603.876,A -85,B 0,C 180,E1 -14662.749,E2 -14662.749} C_VEL
LIN {X 0,Y 333.812,Z 603.901,A -85,B 0,C 180,E1 -14665.17,E2 -14665.17} C_VEL
LIN {X 0,Y 334.108,Z 603.863,A -85,B 0,C 180,E1 -14667.59,E2 -14667.59} C_VEL
LIN {X 0,Y 334.247,Z 603.847,A -85,B 0,C 180,E1 -14670.001,E2 -14670.001} C_VEL
LIN {X 0,Y 334.133,Z 603.865,A -85,B 0,C 180,E1 -14672.412,E2 -14672.412} C_VEL
LIN {X 0,Y 334.028,Z 603.875,A -85,B 0,C 180,E1 -14677.254,E2 -14677.254} C_VEL
LIN {X 0,Y 333.836,Z 603.902,A -85,B 0,C 180,E1 -14680.923,E2 -14680.923} C_VEL
LIN {X 0,Y 333.811,Z 603.905,A -85,B 0,C 180,E1 -14684.635,E2 -14684.635} C_VEL
LIN {X 0,Y 333.799,Z 603.906,A -85,B 0,C 180,E1 -14688.656,E2 -14688.656} C_VEL
LIN {X 0,Y 333.695,Z 603.915,A -85,B 0,C 180,E1 -14692.279,E2 -14692.279} C_VEL
LIN {X 0,Y 333.738,Z 603.91,A -85,B 0,C 180,E1 -14696.247,E2 -14696.247} C_VEL
LIN {X 0,Y 333.679,Z 603.916,A -85,B 0,C 180,E1 -14699.932,E2 -14699.932} C_VEL
LIN {X 0,Y 333.043,Z 604,A -85,B 0,C 180,E1 -14700.939,E2 -14700.939} C_VEL
LIN {X 0,Y 330.199,Z 604.36,A -85,B 0,C 180,E1 -14702.577,E2 -14702.577} C_VEL
LIN {X 0,Y 327.764,Z 604.665,A -85,B 0,C 180,E1 -14703.905,E2 -14703.905} C_VEL
LIN {X 0,Y 326.709,Z 604.792,A -85,B 0,C 180,E1 -14704.932,E2 -14704.932} C_VEL
LIN {X 0,Y 326.62,Z 604.801,A -85,B 0,C 180,E1 -14705.28,E2 -14705.28} C_VEL
LIN {X 0,Y 326.602,Z 604.799,A -85,B 0,C 180,E1 -14708.613,E2 -14708.613} C_VEL
LIN {X 0,Y 326.58,Z 604.802,A -85,B 0,C 180,E1 -14711.847,E2 -14711.847} C_VEL
LIN {X 0,Y 326.561,Z 604.808,A -85,B 0,C 180,E1 -14715.253,E2 -14715.253} C_VEL
LIN {X 0,Y 326.582,Z 604.802,A -85,B 0,C 180,E1 -14718.87,E2 -14718.87} C_VEL
LIN {X 0,Y 326.632,Z 604.795,A -85,B 0,C 180,E1 -14722.762,E2 -14722.762} C_VEL
LIN {X 0,Y 326.613,Z 604.799,A -85,B 0,C 180,E1 -14725.981,E2 -14725.981} C_VEL
LIN {X 0,Y 326.666,Z 604.791,A -85,B 0,C 180,E1 -14730.342,E2 -14730.342} C_VEL
LIN {X 0,Y 326.695,Z 604.787,A -85,B 0,C 180,E1 -14734.517,E2 -14734.517} C_VEL
LIN {X 0,Y 326.625,Z 604.796,A -85,B 0,C 180,E1 -14738.544,E2 -14738.544} C_VEL
LIN {X 0,Y 326.75,Z 604.781,A -85,B 0,C 180,E1 -14741.178,E2 -14741.178} C_VEL
LIN {X 0,Y 326.769,Z 604.779,A -85,B 0,C 180,E1 -14745.433,E2 -14745.433} C_VEL
LIN {X 0,Y 326.775,Z 604.777,A -85,B 0,C 180,E1 -14748.839,E2 -14748.839} C_VEL
LIN {X 0,Y 326.964,Z 604.755,A -85,B 0,C 180,E1 -14752.59,E2 -14752.59} C_VEL
LIN {X 0,Y 326.78,Z 604.776,A -85,B 0,C 180,E1 -14755.065,E2 -14755.065} C_VEL
LIN {X 0,Y 327.052,Z 604.743,A -85,B 0,C 180,E1 -14757.537,E2 -14757.537} C_VEL
LIN {X 0,Y 327.203,Z 604.728,A -85,B 0,C 180,E1 -14760,E2 -14760} C_VEL
LIN {X 0,Y 327.052,Z 604.746,A -85,B 0,C 180,E1 -14762.463,E2 -14762.463} C_VEL
LIN {X 0,Y 326.996,Z 604.754,A -85,B 0,C 180,E1 -14766.169,E2 -14766.169} C_VEL
LIN {X 0,Y 326.812,Z 604.774,A -85,B 0,C 180,E1 -14769.907,E2 -14769.907} C_VEL
LIN {X 0,Y 326.765,Z 604.778,A -85,B 0,C 180,E1 -14773.685,E2 -14773.685} C_VEL
LIN {X 0,Y 326.67,Z 604.79,A -85,B 0,C 180,E1 -14777.53,E2 -14777.53} C_VEL
LIN {X 0,Y 326.624,Z 604.796,A -85,B 0,C 180,E1 -14781.456,E2 -14781.456} C_VEL
LIN {X 0,Y 326.696,Z 604.787,A -85,B 0,C 180,E1 -14785.483,E2 -14785.483} C_VEL
LIN {X 0,Y 326.667,Z 604.79,A -85,B 0,C 180,E1 -14789.659,E2 -14789.659} C_VEL
LIN {X 0,Y 326.613,Z 604.797,A -85,B 0,C 180,E1 -14794.019,E2 -14794.019} C_VEL
LIN {X 0,Y 326.633,Z 604.797,A -85,B 0,C 180,E1 -14797.238,E2 -14797.238} C_VEL
LIN {X 0,Y 326.584,Z 604.805,A -85,B 0,C 180,E1 -14801.131,E2 -14801.131} C_VEL
LIN {X 0,Y 326.562,Z 604.807,A -85,B 0,C 180,E1 -14804.747,E2 -14804.747} C_VEL
LIN {X 0,Y 326.582,Z 604.801,A -85,B 0,C 180,E1 -14808.154,E2 -14808.154} C_VEL
LIN {X 0,Y 326.603,Z 604.802,A -85,B 0,C 180,E1 -14811.387,E2 -14811.387} C_VEL
LIN {X 0,Y 326.624,Z 604.798,A -85,B 0,C 180,E1 -14814.851,E2 -14814.851} C_VEL
LIN {X 0,Y 326.605,Z 604.86,A -85,B 0,C 180,E1 -14817.169,E2 -14817.169} C_VEL
LIN {X 0,Y 329.633,Z 618.739,A -85,B 0,C 180,E1 -14820.945,E2 -14820.945} C_VEL
LIN {X 0,Y 331.337,Z 627.395,A -85,B 0,C 180,E1 -14823.205,E2 -14823.205} C_VEL
LIN {X 0,Y 329.806,Z 640.831,A -85,B 0,C 180,E1 -14826.393,E2 -14826.393} C_VEL
LIN {X 0,Y 335.095,Z 681.032,A -85,B 0,C 180,E1 -14827.747,E2 -14827.747} C_VEL
LIN {X 0,Y 333.502,Z 750.075,A -85,B 0,C 180,E1 -14829.45,E2 -14829.45} C_VEL
LIN {X 0,Y 332.727,Z 764.113,A -85,B 0,C 180,E1 -14830.045,E2 -14830.045} C_VEL
LIN {X 0,Y 331.681,Z 776.677,A -85,B 0,C 180,E1 -14830.825,E2 -14830.825} C_VEL
LIN {X 0,Y 330.572,Z 789.165,A -85,B 0,C 180,E1 -14831.883,E2 -14831.883} C_VEL
LIN {X 0,Y 329.336,Z 800.366,A -85,B 0,C 180,E1 -14833.095,E2 -14833.095} C_VEL
LIN {X 0,Y 328.35,Z 810.014,A -85,B 0,C 180,E1 -14834.404,E2 -14834.404} C_VEL
LIN {X 0,Y 327.319,Z 819.664,A -85,B 0,C 180,E1 -14836.02,E2 -14836.02} C_VEL
LIN {X 0,Y 326.376,Z 828.614,A -85,B 0,C 180,E1 -14837.879,E2 -14837.879} C_VEL
LIN {X 0,Y 325.684,Z 835.727,A -85,B 0,C 180,E1 -14839.744,E2 -14839.744} C_VEL
LIN {X 0,Y 325.233,Z 842.228,A -85,B 0,C 180,E1 -14841.924,E2 -14841.924} C_VEL
LIN {X 0,Y 325.072,Z 846.868,A -85,B 0,C 180,E1 -14843.997,E2 -14843.997} C_VEL
LIN {X 0,Y 325.038,Z 848.664,A -85,B 0,C 180,E1 -14845.037,E2 -14845.037} C_VEL
LIN {X 0,Y 325.006,Z 850.365,A -85,B 0,C 180,E1 -14846.279,E2 -14846.279} C_VEL
LIN {X 0,Y 325.027,Z 851.644,A -85,B 0,C 180,E1 -14847.52,E2 -14847.52} C_VEL
LIN {X 0,Y 325.148,Z 852.509,A -85,B 0,C 180,E1 -14848.76,E2 -14848.76} C_VEL
LIN {X 0,Y 325.192,Z 852.907,A -85,B 0,C 180,E1 -14849.999,E2 -14849.999} C_VEL
LIN {X 0,Y 325.11,Z 852.875,A -85,B 0,C 180,E1 -14851.237,E2 -14851.237} C_VEL
LIN {X 0,Y 324.99,Z 852.435,A -85,B 0,C 180,E1 -14852.477,E2 -14852.477} C_VEL
LIN {X 0,Y 324.982,Z 851.591,A -85,B 0,C 180,E1 -14853.718,E2 -14853.718} C_VEL
LIN {X 0,Y 324.999,Z 849.062,A -85,B 0,C 180,E1 -14855.879,E2 -14855.879} C_VEL
LIN {X 0,Y 325.227,Z 845.117,A -85,B 0,C 180,E1 -14858.073,E2 -14858.073} C_VEL
LIN {X 0,Y 325.653,Z 840.583,A -85,B 0,C 180,E1 -14859.94,E2 -14859.94} C_VEL
LIN {X 0,Y 326.453,Z 833.783,A -85,B 0,C 180,E1 -14862.115,E2 -14862.115} C_VEL
LIN {X 0,Y 327.619,Z 826.378,A -85,B 0,C 180,E1 -14863.964,E2 -14863.964} C_VEL
LIN {X 0,Y 328.873,Z 817.608,A -85,B 0,C 180,E1 -14865.736,E2 -14865.736} C_VEL
LIN {X 0,Y 330.262,Z 807.875,A -85,B 0,C 180,E1 -14867.331,E2 -14867.331} C_VEL
LIN {X 0,Y 331.733,Z 797.547,A -85,B 0,C 180,E1 -14868.688,E2 -14868.688} C_VEL
LIN {X 0,Y 333.344,Z 786.181,A -85,B 0,C 180,E1 -14869.873,E2 -14869.873} C_VEL
LIN {X 0,Y 334.599,Z 775.517,A -85,B 0,C 180,E1 -14870.758,E2 -14870.758} C_VEL
LIN {X 0,Y 335.937,Z 762.822,A -85,B 0,C 180,E1 -14871.555,E2 -14871.555} C_VEL
LIN {X 0,Y 336.935,Z 749.654,A -85,B 0,C 180,E1 -14872.13,E2 -14872.13} C_VEL
LIN {X 0,Y 337.682,Z 728.485,A -85,B 0,C 180,E1 -14872.707,E2 -14872.707} C_VEL
LIN {X 0,Y 339.137,Z 681.604,A -85,B 0,C 180,E1 -14873.893,E2 -14873.893} C_VEL
LIN {X 0,Y 336.566,Z 661.54,A -85,B 0,C 180,E1 -14874.72,E2 -14874.72} C_VEL
LIN {X 0,Y 333.057,Z 642.825,A -85,B 0,C 180,E1 -14875.636,E2 -14875.636} C_VEL
LIN {X 0,Y 331.923,Z 637.372,A -85,B 0,C 180,E1 -14875.943,E2 -14875.943} C_VEL
LIN {X 0,Y 332.661,Z 631.396,A -85,B 0,C 180,E1 -14877.461,E2 -14877.461} C_VEL
LIN {X 0,Y 331.059,Z 622.766,A -85,B 0,C 180,E1 -14879.992,E2 -14879.992} C_VEL
LIN {X 0,Y 328.522,Z 611.935,A -85,B 0,C 180,E1 -14883.455,E2 -14883.455} C_VEL
LIN {X 0,Y 326.627,Z 604.8,A -85,B 0,C 180,E1 -14885.991,E2 -14885.991} C_VEL
LIN {X 0,Y 326.63,Z 604.8,A -85,B 0,C 180,E1 -14889.231,E2 -14889.231} C_VEL
LIN {X 0,Y 326.61,Z 604.805,A -85,B 0,C 180,E1 -14893.515,E2 -14893.515} C_VEL
LIN {X 0,Y 326.628,Z 604.799,A -85,B 0,C 180,E1 -14897.016,E2 -14897.016} C_VEL
LIN {X 0,Y 326.64,Z 604.795,A -85,B 0,C 180,E1 -14900.764,E2 -14900.764} C_VEL
LIN {X 0,Y 326.608,Z 604.802,A -85,B 0,C 180,E1 -14904.479,E2 -14904.479} C_VEL
LIN {X 0,Y 326.609,Z 604.799,A -85,B 0,C 180,E1 -14907.455,E2 -14907.455} C_VEL
LIN {X 0,Y 326.655,Z 604.792,A -85,B 0,C 180,E1 -14910.34,E2 -14910.34} C_VEL
LIN {X 0,Y 326.683,Z 604.787,A -85,B 0,C 180,E1 -14914.515,E2 -14914.515} C_VEL
LIN {X 0,Y 326.639,Z 604.797,A -85,B 0,C 180,E1 -14918.545,E2 -14918.545} C_VEL
LIN {X 0,Y 326.736,Z 604.785,A -85,B 0,C 180,E1 -14921.177,E2 -14921.177} C_VEL
LIN {X 0,Y 326.755,Z 604.778,A -85,B 0,C 180,E1 -14925.432,E2 -14925.432} C_VEL
LIN {X 0,Y 326.765,Z 604.783,A -85,B 0,C 180,E1 -14928.839,E2 -14928.839} C_VEL
LIN {X 0,Y 326.971,Z 604.754,A -85,B 0,C 180,E1 -14932.59,E2 -14932.59} C_VEL
LIN {X 0,Y 326.772,Z 604.779,A -85,B 0,C 180,E1 -14935.065,E2 -14935.065} C_VEL
LIN {X 0,Y 327.04,Z 604.747,A -85,B 0,C 180,E1 -14937.537,E2 -14937.537} C_VEL
LIN {X 0,Y 327.21,Z 604.728,A -85,B 0,C 180,E1 -14940,E2 -14940} C_VEL
LIN {X 0,Y 327.061,Z 604.746,A -85,B 0,C 180,E1 -14942.463,E2 -14942.463} C_VEL
LIN {X 0,Y 326.991,Z 604.842,A -85,B 0,C 180,E1 -14947.138,E2 -14947.138} C_VEL
LIN {X 0,Y 327.817,Z 608.659,A -85,B 0,C 180,E1 -14948.703,E2 -14948.703} C_VEL
LIN {X 0,Y 336.882,Z 627.359,A -85,B 0,C 180,E1 -14950.28,E2 -14950.28} C_VEL
LIN {X 0,Y 340.444,Z 636.076,A -85,B 0,C 180,E1 -14950.894,E2 -14950.894} C_VEL
LIN {X 0,Y 337.748,Z 714.383,A -85,B 0,C 180,E1 -14952.906,E2 -14952.906} C_VEL
LIN {X 0,Y 336.982,Z 727.824,A -85,B 0,C 180,E1 -14953.493,E2 -14953.493} C_VEL
LIN {X 0,Y 335.995,Z 740.576,A -85,B 0,C 180,E1 -14954.305,E2 -14954.305} C_VEL
LIN {X 0,Y 334.748,Z 753.026,A -85,B 0,C 180,E1 -14955.382,E2 -14955.382} C_VEL
LIN {X 0,Y 333.477,Z 763.496,A -85,B 0,C 180,E1 -14956.53,E2 -14956.53} C_VEL
LIN {X 0,Y 332.127,Z 772.843,A -85,B 0,C 180,E1 -14957.787,E2 -14957.787} C_VEL
LIN {X 0,Y 330.779,Z 781.567,A -85,B 0,C 180,E1 -14959.228,E2 -14959.228} C_VEL
LIN {X 0,Y 329.367,Z 790.282,A -85,B 0,C 180,E1 -14961.014,E2 -14961.014} C_VEL
LIN {X 0,Y 328.081,Z 797.698,A -85,B 0,C 180,E1 -14962.913,E2 -14962.913} C_VEL
LIN {X 0,Y 327.206,Z 803.35,A -85,B 0,C 180,E1 -14964.752,E2 -14964.752} C_VEL
LIN {X 0,Y 326.354,Z 808.365,A -85,B 0,C 180,E1 -14966.887,E2 -14966.887} C_VEL
LIN {X 0,Y 325.888,Z 810.954,A -85,B 0,C 180,E1 -14968.323,E2 -14968.323} C_VEL
LIN {X 0,Y 325.415,Z 813.461,A -85,B 0,C 180,E1 -14970.248,E2 -14970.248} C_VEL
LIN {X 0,Y 325.054,Z 815.092,A -85,B 0,C 180,E1 -14972.521,E2 -14972.521} C_VEL
LIN {X 0,Y 324.899,Z 815.347,A -85,B 0,C 180,E1 -14974.718,E2 -14974.718} C_VEL
LIN {X 0,Y 324.905,Z 814.382,A -85,B 0,C 180,E1 -14976.84,E2 -14976.84} C_VEL
LIN {X 0,Y 325.097,Z 812.28,A -85,B 0,C 180,E1 -14978.902,E2 -14978.902} C_VEL
LIN {X 0,Y 325.475,Z 809.073,A -85,B 0,C 180,E1 -14980.911,E2 -14980.911} C_VEL
LIN {X 0,Y 325.818,Z 804.853,A -85,B 0,C 180,E1 -14982.831,E2 -14982.831} C_VEL
LIN {X 0,Y 326.395,Z 799.435,A -85,B 0,C 180,E1 -14984.722,E2 -14984.722} C_VEL
LIN {X 0,Y 327.127,Z 792.742,A -85,B 0,C 180,E1 -14986.571,E2 -14986.571} C_VEL
LIN {X 0,Y 328.05,Z 784.562,A -85,B 0,C 180,E1 -14988.386,E2 -14988.386} C_VEL
LIN {X 0,Y 329.06,Z 775.73,A -85,B 0,C 180,E1 -14989.976,E2 -14989.976} C_VEL
LIN {X 0,Y 330.155,Z 765.409,A -85,B 0,C 180,E1 -14991.471,E2 -14991.471} C_VEL
LIN {X 0,Y 331.177,Z 754.626,A -85,B 0,C 180,E1 -14992.73,E2 -14992.73} C_VEL
LIN {X 0,Y 332.163,Z 743.602,A -85,B 0,C 180,E1 -14993.753,E2 -14993.753} C_VEL
LIN {X 0,Y 332.991,Z 731.57,A -85,B 0,C 180,E1 -14994.614,E2 -14994.614} C_VEL
LIN {X 0,Y 333.585,Z 718.222,A -85,B 0,C 180,E1 -14995.304,E2 -14995.304} C_VEL
LIN {X 0,Y 334.022,Z 705.384,A -85,B 0,C 180,E1 -14995.727,E2 -14995.727} C_VEL
LIN {X 0,Y 335.952,Z 631.843,A -85,B 0,C 180,E1 -14997.497,E2 -14997.497} C_VEL
LIN {X 0,Y 330.107,Z 614.503,A -85,B 0,C 180,E1 -14998.301,E2 -14998.301} C_VEL
LIN {X 0,Y 326.63,Z 604.796,A -85,B 0,C 180,E1 -14998.798,E2 -14998.798} C_VEL
LIN {X 0,Y 326.653,Z 604.797,A -85,B 0,C 180,E1 -15001.899,E2 -15001.899} C_VEL
LIN {X 0,Y 326.685,Z 604.789,A -85,B 0,C 180,E1 -15004.629,E2 -15004.629} C_VEL
LIN {X 0,Y 326.65,Z 604.795,A -85,B 0,C 180,E1 -15008.547,E2 -15008.547} C_VEL
LIN {X 0,Y 326.742,Z 604.781,A -85,B 0,C 180,E1 -15011.179,E2 -15011.179} C_VEL
LIN {X 0,Y 326.762,Z 604.779,A -85,B 0,C 180,E1 -15015.434,E2 -15015.434} C_VEL
LIN {X 0,Y 326.773,Z 604.779,A -85,B 0,C 180,E1 -15018.84,E2 -15018.84} C_VEL
LIN {X 0,Y 326.98,Z 604.756,A -85,B 0,C 180,E1 -15022.592,E2 -15022.592} C_VEL
LIN {X 0,Y 326.779,Z 604.777,A -85,B 0,C 180,E1 -15025.066,E2 -15025.066} C_VEL
LIN {X 0,Y 327.049,Z 604.743,A -85,B 0,C 180,E1 -15027.538,E2 -15027.538} C_VEL
LIN {X 0,Y 327.198,Z 604.725,A -85,B 0,C 180,E1 -15030.001,E2 -15030.001} C_VEL
LIN {X 0,Y 327.07,Z 604.745,A -85,B 0,C 180,E1 -15032.464,E2 -15032.464} C_VEL
LIN {X 0,Y 326.998,Z 604.751,A -85,B 0,C 180,E1 -15036.17,E2 -15036.17} C_VEL
LIN {X 0,Y 326.916,Z 604.765,A -85,B 0,C 180,E1 -15038.656,E2 -15038.656} C_VEL
LIN {X 0,Y 326.737,Z 604.784,A -85,B 0,C 180,E1 -15042.422,E2 -15042.422} C_VEL
LIN {X 0,Y 326.757,Z 604.784,A -85,B 0,C 180,E1 -15044.959,E2 -15044.959} C_VEL
LIN {X 0,Y 326.735,Z 604.788,A -85,B 0,C 180,E1 -15048.839,E2 -15048.839} C_VEL
LIN {X 0,Y 326.624,Z 604.8,A -85,B 0,C 180,E1 -15052.788,E2 -15052.788} C_VEL
LIN {X 0,Y 326.693,Z 604.789,A -85,B 0,C 180,E1 -15055.485,E2 -15055.485} C_VEL
LIN {X 0,Y 326.651,Z 604.793,A -85,B 0,C 180,E1 -15059.661,E2 -15059.661} C_VEL
LIN {X 0,Y 326.611,Z 604.797,A -85,B 0,C 180,E1 -15064.02,E2 -15064.02} C_VEL
LIN {X 0,Y 326.62,Z 604.801,A -85,B 0,C 180,E1 -15065.28,E2 -15065.28} C_VEL
LIN {X 0,Y 325.935,Z 604.883,A -85,B 0,C 180,E1 -15066.308,E2 -15066.308} C_VEL
LIN {X 0,Y 323.054,Z 605.241,A -85,B 0,C 180,E1 -15067.98,E2 -15067.98} C_VEL
LIN {X 0,Y 320.626,Z 605.548,A -85,B 0,C 180,E1 -15069.335,E2 -15069.335} C_VEL
LIN {X 0,Y 319.594,Z 605.672,A -85,B 0,C 180,E1 -15070.384,E2 -15070.384} C_VEL
LIN {X 0,Y 319.514,Z 605.682,A -85,B 0,C 180,E1 -15070.74,E2 -15070.74} C_VEL
LIN {X 0,Y 319.56,Z 605.68,A -85,B 0,C 180,E1 -15073.468,E2 -15073.468} C_VEL
LIN {X 0,Y 319.566,Z 605.677,A -85,B 0,C 180,E1 -15077.019,E2 -15077.019} C_VEL
LIN {X 0,Y 319.551,Z 605.676,A -85,B 0,C 180,E1 -15080.372,E2 -15080.372} C_VEL
LIN {X 0,Y 319.563,Z 605.68,A -85,B 0,C 180,E1 -15083.573,E2 -15083.573} C_VEL
LIN {X 0,Y 319.582,Z 605.672,A -85,B 0,C 180,E1 -15086.687,E2 -15086.687} C_VEL
LIN {X 0,Y 319.597,Z 605.677,A -85,B 0,C 180,E1 -15089.617,E2 -15089.617} C_VEL
LIN {X 0,Y 319.614,Z 605.669,A -85,B 0,C 180,E1 -15092.499,E2 -15092.499} C_VEL
LIN {X 0,Y 319.608,Z 605.672,A -85,B 0,C 180,E1 -15095.304,E2 -15095.304} C_VEL
LIN {X 0,Y 319.608,Z 605.672,A -85,B 0,C 180,E1 -15099.401,E2 -15099.401} C_VEL
LIN {X 0,Y 319.664,Z 605.666,A -85,B 0,C 180,E1 -15102.074,E2 -15102.074} C_VEL
LIN {X 0,Y 319.738,Z 605.658,A -85,B 0,C 180,E1 -15106.008,E2 -15106.008} C_VEL
LIN {X 0,Y 319.758,Z 605.655,A -85,B 0,C 180,E1 -15109.873,E2 -15109.873} C_VEL
LIN {X 0,Y 319.918,Z 605.633,A -85,B 0,C 180,E1 -15112.426,E2 -15112.426} C_VEL
LIN {X 0,Y 319.75,Z 605.652,A -85,B 0,C 180,E1 -15114.956,E2 -15114.956} C_VEL
LIN {X 0,Y 319.995,Z 605.622,A -85,B 0,C 180,E1 -15117.483,E2 -15117.483} C_VEL
LIN {X 0,Y 320.155,Z 605.605,A -85,B 0,C 180,E1 -15120,E2 -15120} C_VEL
LIN {X 0,Y 319.996,Z 605.624,A -85,B 0,C 180,E1 -15122.518,E2 -15122.518} C_VEL
LIN {X 0,Y 319.95,Z 605.633,A -85,B 0,C 180,E1 -15126.306,E2 -15126.306} C_VEL
LIN {X 0,Y 319.843,Z 605.642,A -85,B 0,C 180,E1 -15128.848,E2 -15128.848} C_VEL
LIN {X 0,Y 319.688,Z 605.663,A -85,B 0,C 180,E1 -15132.7,E2 -15132.7} C_VEL
LIN {X 0,Y 319.685,Z 605.66,A -85,B 0,C 180,E1 -15135.296,E2 -15135.296} C_VEL
LIN {X 0,Y 319.594,Z 605.672,A -85,B 0,C 180,E1 -15139.26,E2 -15139.26} C_VEL
LIN {X 0,Y 319.566,Z 605.675,A -85,B 0,C 180,E1 -15143.32,E2 -15143.32} C_VEL
LIN {X 0,Y 319.641,Z 605.667,A -85,B 0,C 180,E1 -15146.088,E2 -15146.088} C_VEL
LIN {X 0,Y 319.596,Z 605.675,A -85,B 0,C 180,E1 -15148.933,E2 -15148.933} C_VEL
LIN {X 0,Y 319.538,Z 605.678,A -85,B 0,C 180,E1 -15151.861,E2 -15151.861} C_VEL
LIN {X 0,Y 319.585,Z 605.673,A -85,B 0,C 180,E1 -15155.542,E2 -15155.542} C_VEL
LIN {X 0,Y 319.564,Z 605.676,A -85,B 0,C 180,E1 -15159.668,E2 -15159.668} C_VEL
LIN {X 0,Y 319.563,Z 605.677,A -85,B 0,C 180,E1 -15163.467,E2 -15163.467} C_VEL
LIN {X 0,Y 319.566,Z 605.681,A -85,B 0,C 180,E1 -15167.017,E2 -15167.017} C_VEL
LIN {X 0,Y 319.552,Z 605.677,A -85,B 0,C 180,E1 -15170.37,E2 -15170.37} C_VEL
LIN {X 0,Y 319.585,Z 605.673,A -85,B 0,C 180,E1 -15174.456,E2 -15174.456} C_VEL
LIN {X 0,Y 319.589,Z 605.771,A -85,B 0,C 180,E1 -15176.833,E2 -15176.833} C_VEL
LIN {X 0,Y 322.686,Z 620.164,A -85,B 0,C 180,E1 -15180.836,E2 -15180.836} C_VEL
LIN {X 0,Y 324.26,Z 627.974,A -85,B 0,C 180,E1 -15182.924,E2 -15182.924} C_VEL
LIN {X 0,Y 323.982,Z 632.106,A -85,B 0,C 180,E1 -15183.941,E2 -15183.941} C_VEL
LIN {X 0,Y 322.956,Z 640.434,A -85,B 0,C 180,E1 -15185.958,E2 -15185.958} C_VEL
LIN {X 0,Y 328.378,Z 682.919,A -85,B 0,C 180,E1 -15187.429,E2 -15187.429} C_VEL
LIN {X 0,Y 326.658,Z 750.028,A -85,B 0,C 180,E1 -15189.123,E2 -15189.123} C_VEL
LIN {X 0,Y 325.875,Z 763.94,A -85,B 0,C 180,E1 -15189.731,E2 -15189.731} C_VEL
LIN {X 0,Y 324.867,Z 775.934,A -85,B 0,C 180,E1 -15190.489,E2 -15190.489} C_VEL
LIN {X 0,Y 323.714,Z 787.678,A -85,B 0,C 180,E1 -15191.486,E2 -15191.486} C_VEL
LIN {X 0,Y 322.444,Z 799.076,A -85,B 0,C 180,E1 -15192.723,E2 -15192.723} C_VEL
LIN {X 0,Y 321.456,Z 808.892,A -85,B 0,C 180,E1 -15194.056,E2 -15194.056} C_VEL
LIN {X 0,Y 320.4,Z 818.708,A -85,B 0,C 180,E1 -15195.712,E2 -15195.712} C_VEL
LIN {X 0,Y 319.395,Z 827.755,A -85,B 0,C 180,E1 -15197.61,E2 -15197.61} C_VEL
LIN {X 0,Y 318.657,Z 834.983,A -85,B 0,C 180,E1 -15199.515,E2 -15199.515} C_VEL
LIN {X 0,Y 318.18,Z 841.553,A -85,B 0,C 180,E1 -15201.744,E2 -15201.744} C_VEL
LIN {X 0,Y 318.011,Z 845.847,A -85,B 0,C 180,E1 -15203.655,E2 -15203.655} C_VEL
LIN {X 0,Y 317.964,Z 848.1,A -85,B 0,C 180,E1 -15204.926,E2 -15204.926} C_VEL
LIN {X 0,Y 317.935,Z 849.837,A -85,B 0,C 180,E1 -15206.196,E2 -15206.196} C_VEL
LIN {X 0,Y 317.937,Z 851.139,A -85,B 0,C 180,E1 -15207.465,E2 -15207.465} C_VEL
LIN {X 0,Y 318.055,Z 852.03,A -85,B 0,C 180,E1 -15208.732,E2 -15208.732} C_VEL
LIN {X 0,Y 318.117,Z 852.475,A -85,B 0,C 180,E1 -15209.999,E2 -15209.999} C_VEL
LIN {X 0,Y 318.014,Z 852.464,A -85,B 0,C 180,E1 -15211.265,E2 -15211.265} C_VEL
LIN {X 0,Y 317.906,Z 851.225,A -85,B 0,C 180,E1 -15213.801,E2 -15213.801} C_VEL
LIN {X 0,Y 317.894,Z 849.033,A -85,B 0,C 180,E1 -15215.808,E2 -15215.808} C_VEL
LIN {X 0,Y 318.06,Z 846.109,A -85,B 0,C 180,E1 -15217.617,E2 -15217.617} C_VEL
LIN {X 0,Y 318.437,Z 842.011,A -85,B 0,C 180,E1 -15219.526,E2 -15219.526} C_VEL
LIN {X 0,Y 319.182,Z 835.765,A -85,B 0,C 180,E1 -15221.75,E2 -15221.75} C_VEL
LIN {X 0,Y 320.273,Z 828.943,A -85,B 0,C 180,E1 -15223.643,E2 -15223.643} C_VEL
LIN {X 0,Y 321.491,Z 820.982,A -85,B 0,C 180,E1 -15225.432,E2 -15225.432} C_VEL
LIN {X 0,Y 322.844,Z 811.939,A -85,B 0,C 180,E1 -15227.089,E2 -15227.089} C_VEL
LIN {X 0,Y 324.505,Z 801.445,A -85,B 0,C 180,E1 -15228.628,E2 -15228.628} C_VEL
LIN {X 0,Y 326.325,Z 789.75,A -85,B 0,C 180,E1 -15229.991,E2 -15229.991} C_VEL
LIN {X 0,Y 327.741,Z 778.313,A -85,B 0,C 180,E1 -15231.048,E2 -15231.048} C_VEL
LIN {X 0,Y 329.267,Z 765.418,A -85,B 0,C 180,E1 -15231.932,E2 -15231.932} C_VEL
LIN {X 0,Y 330.406,Z 752.029,A -85,B 0,C 180,E1 -15232.593,E2 -15232.593} C_VEL
LIN {X 0,Y 331.057,Z 737.603,A -85,B 0,C 180,E1 -15233.041,E2 -15233.041} C_VEL
LIN {X 0,Y 332.91,Z 682.264,A -85,B 0,C 180,E1 -15234.468,E2 -15234.468} C_VEL
LIN {X 0,Y 330.434,Z 662.842,A -85,B 0,C 180,E1 -15235.304,E2 -15235.304} C_VEL
LIN {X 0,Y 327.273,Z 645.43,A -85,B 0,C 180,E1 -15236.182,E2 -15236.182} C_VEL
LIN {X 0,Y 325.455,Z 636.849,A -85,B 0,C 180,E1 -15236.68,E2 -15236.68} C_VEL
LIN {X 0,Y 325.802,Z 632.573,A -85,B 0,C 180,E1 -15237.818,E2 -15237.818} C_VEL
LIN {X 0,Y 324.018,Z 623.304,A -85,B 0,C 180,E1 -15240.643,E2 -15240.643} C_VEL
LIN {X 0,Y 321.69,Z 613.568,A -85,B 0,C 180,E1 -15243.881,E2 -15243.881} C_VEL
LIN {X 0,Y 319.601,Z 605.677,A -85,B 0,C 180,E1 -15246.812,E2 -15246.812} C_VEL
LIN {X 0,Y 319.56,Z 605.683,A -85,B 0,C 180,E1 -15249.669,E2 -15249.669} C_VEL
LIN {X 0,Y 319.587,Z 605.68,A -85,B 0,C 180,E1 -15253.473,E2 -15253.473} C_VEL
LIN {X 0,Y 319.604,Z 605.674,A -85,B 0,C 180,E1 -15257.024,E2 -15257.024} C_VEL
LIN {X 0,Y 319.58,Z 605.677,A -85,B 0,C 180,E1 -15260.375,E2 -15260.375} C_VEL
LIN {X 0,Y 319.555,Z 605.675,A -85,B 0,C 180,E1 -15263.572,E2 -15263.572} C_VEL
LIN {X 0,Y 319.572,Z 605.675,A -85,B 0,C 180,E1 -15266.685,E2 -15266.685} C_VEL
LIN {X 0,Y 319.587,Z 605.672,A -85,B 0,C 180,E1 -15269.616,E2 -15269.616} C_VEL
LIN {X 0,Y 319.603,Z 605.672,A -85,B 0,C 180,E1 -15272.497,E2 -15272.497} C_VEL
LIN {X 0,Y 319.598,Z 605.672,A -85,B 0,C 180,E1 -15275.303,E2 -15275.303} C_VEL
LIN {X 0,Y 319.589,Z 605.675,A -85,B 0,C 180,E1 -15278.047,E2 -15278.047} C_VEL
LIN {X 0,Y 319.681,Z 605.665,A -85,B 0,C 180,E1 -15280.961,E2 -15280.961} C_VEL
LIN {X 0,Y 319.723,Z 605.654,A -85,B 0,C 180,E1 -15285.275,E2 -15285.275} C_VEL
LIN {X 0,Y 319.751,Z 605.654,A -85,B 0,C 180,E1 -15289.872,E2 -15289.872} C_VEL
LIN {X 0,Y 319.925,Z 605.632,A -85,B 0,C 180,E1 -15292.426,E2 -15292.426} C_VEL
LIN {X 0,Y 319.741,Z 605.655,A -85,B 0,C 180,E1 -15294.956,E2 -15294.956} C_VEL
LIN {X 0,Y 319.984,Z 605.626,A -85,B 0,C 180,E1 -15297.482,E2 -15297.482} C_VEL
LIN {X 0,Y 320.161,Z 605.606,A -85,B 0,C 180,E1 -15300,E2 -15300} C_VEL
LIN {X 0,Y 320.002,Z 605.625,A -85,B 0,C 180,E1 -15302.517,E2 -15302.517} C_VEL
LIN {X 0,Y 319.957,Z 605.823,A -85,B 0,C 180,E1 -15306.384,E2 -15306.384} C_VEL
LIN {X 0,Y 320.813,Z 609.252,A -85,B 0,C 180,E1 -15307.869,E2 -15307.869} C_VEL
LIN {X 0,Y 329.668,Z 627.042,A -85,B 0,C 180,E1 -15309.493,E2 -15309.493} C_VEL
LIN {X 0,Y 334.281,Z 637.979,A -85,B 0,C 180,E1 -15310.328,E2 -15310.328} C_VEL
LIN {X 0,Y 331.465,Z 714.681,A -85,B 0,C 180,E1 -15312.345,E2 -15312.345} C_VEL
LIN {X 0,Y 330.643,Z 728.355,A -85,B 0,C 180,E1 -15312.951,E2 -15312.951} C_VEL
LIN {X 0,Y 329.59,Z 741.373,A -85,B 0,C 180,E1 -15313.801,E2 -15313.801} C_VEL
LIN {X 0,Y 328.293,Z 753.647,A -85,B 0,C 180,E1 -15314.886,E2 -15314.886} C_VEL
LIN {X 0,Y 326.926,Z 764.369,A -85,B 0,C 180,E1 -15316.093,E2 -15316.093} C_VEL
LIN {X 0,Y 325.426,Z 774.013,A -85,B 0,C 180,E1 -15317.436,E2 -15317.436} C_VEL
LIN {X 0,Y 323.947,Z 783.015,A -85,B 0,C 180,E1 -15318.991,E2 -15318.991} C_VEL
LIN {X 0,Y 322.543,Z 791.089,A -85,B 0,C 180,E1 -15320.703,E2 -15320.703} C_VEL
LIN {X 0,Y 321.31,Z 797.794,A -85,B 0,C 180,E1 -15322.455,E2 -15322.455} C_VEL
LIN {X 0,Y 320.477,Z 802.415,A -85,B 0,C 180,E1 -15323.935,E2 -15323.935} C_VEL
LIN {X 0,Y 319.547,Z 807.772,A -85,B 0,C 180,E1 -15326.096,E2 -15326.096} C_VEL
LIN {X 0,Y 318.871,Z 811.542,A -85,B 0,C 180,E1 -15328.166,E2 -15328.166} C_VEL
LIN {X 0,Y 318.288,Z 814.36,A -85,B 0,C 180,E1 -15330.558,E2 -15330.558} C_VEL
LIN {X 0,Y 317.931,Z 815.683,A -85,B 0,C 180,E1 -15332.862,E2 -15332.862} C_VEL
LIN {X 0,Y 317.81,Z 815.683,A -85,B 0,C 180,E1 -15335.097,E2 -15335.097} C_VEL
LIN {X 0,Y 317.846,Z 814.461,A -85,B 0,C 180,E1 -15337.252,E2 -15337.252} C_VEL
LIN {X 0,Y 318.086,Z 812.09,A -85,B 0,C 180,E1 -15339.35,E2 -15339.35} C_VEL
LIN {X 0,Y 318.468,Z 808.487,A -85,B 0,C 180,E1 -15341.456,E2 -15341.456} C_VEL
LIN {X 0,Y 318.867,Z 804.142,A -85,B 0,C 180,E1 -15343.339,E2 -15343.339} C_VEL
LIN {X 0,Y 319.498,Z 798.451,A -85,B 0,C 180,E1 -15345.261,E2 -15345.261} C_VEL
LIN {X 0,Y 320.278,Z 791.487,A -85,B 0,C 180,E1 -15347.139,E2 -15347.139} C_VEL
LIN {X 0,Y 321.316,Z 782.872,A -85,B 0,C 180,E1 -15348.993,E2 -15348.993} C_VEL
LIN {X 0,Y 322.415,Z 773.487,A -85,B 0,C 180,E1 -15350.619,E2 -15350.619} C_VEL
LIN {X 0,Y 323.523,Z 763.125,A -85,B 0,C 180,E1 -15352.077,E2 -15352.077} C_VEL
LIN {X 0,Y 324.658,Z 751.362,A -85,B 0,C 180,E1 -15353.383,E2 -15353.383} C_VEL
LIN {X 0,Y 325.684,Z 739.197,A -85,B 0,C 180,E1 -15354.434,E2 -15354.434} C_VEL
LIN {X 0,Y 326.43,Z 726.723,A -85,B 0,C 180,E1 -15355.244,E2 -15355.244} C_VEL
LIN {X 0,Y 327.002,Z 712.942,A -85,B 0,C 180,E1 -15355.857,E2 -15355.857} C_VEL
LIN {X 0,Y 329.148,Z 632.666,A -85,B 0,C 180,E1 -15357.875,E2 -15357.875} C_VEL
LIN {X 0,Y 321.277,Z 610.398,A -85,B 0,C 180,E1 -15358.968,E2 -15358.968} C_VEL
LIN {X 0,Y 319.603,Z 605.672,A -85,B 0,C 180,E1 -15359.225,E2 -15359.225} C_VEL
LIN {X 0,Y 319.602,Z 605.672,A -85,B 0,C 180,E1 -15362.499,E2 -15362.499} C_VEL
LIN {X 0,Y 319.602,Z 605.671,A -85,B 0,C 180,E1 -15365.305,E2 -15365.305} C_VEL
LIN {X 0,Y 319.62,Z 605.669,A -85,B 0,C 180,E1 -15369.403,E2 -15369.403} C_VEL
LIN {X 0,Y 319.657,Z 605.668,A -85,B 0,C 180,E1 -15372.075,E2 -15372.075} C_VEL
LIN {X 0,Y 319.732,Z 605.658,A -85,B 0,C 180,E1 -15376.009,E2 -15376.009} C_VEL
LIN {X 0,Y 319.759,Z 605.652,A -85,B 0,C 180,E1 -15379.874,E2 -15379.874} C_VEL
LIN {X 0,Y 319.933,Z 605.635,A -85,B 0,C 180,E1 -15382.428,E2 -15382.428} C_VEL
LIN {X 0,Y 319.749,Z 605.654,A -85,B 0,C 180,E1 -15384.958,E2 -15384.958} C_VEL
LIN {X 0,Y 319.993,Z 605.622,A -85,B 0,C 180,E1 -15387.484,E2 -15387.484} C_VEL
LIN {X 0,Y 320.15,Z 605.603,A -85,B 0,C 180,E1 -15390.001,E2 -15390.001} C_VEL
LIN {X 0,Y 320.01,Z 605.625,A -85,B 0,C 180,E1 -15392.519,E2 -15392.519} C_VEL
LIN {X 0,Y 319.954,Z 605.629,A -85,B 0,C 180,E1 -15396.307,E2 -15396.307} C_VEL
LIN {X 0,Y 319.844,Z 605.645,A -85,B 0,C 180,E1 -15398.849,E2 -15398.849} C_VEL
LIN {X 0,Y 319.685,Z 605.665,A -85,B 0,C 180,E1 -15402.701,E2 -15402.701} C_VEL
LIN {X 0,Y 319.702,Z 605.66,A -85,B 0,C 180,E1 -15405.297,E2 -15405.297} C_VEL
LIN {X 0,Y 319.677,Z 605.663,A -85,B 0,C 180,E1 -15409.256,E2 -15409.256} C_VEL
LIN {X 0,Y 319.573,Z 605.677,A -85,B 0,C 180,E1 -15413.32,E2 -15413.32} C_VEL
LIN {X 0,Y 319.621,Z 605.668,A -85,B 0,C 180,E1 -15416.091,E2 -15416.091} C_VEL
LIN {X 0,Y 319.584,Z 605.677,A -85,B 0,C 180,E1 -15418.936,E2 -15418.936} C_VEL
LIN {X 0,Y 319.534,Z 605.679,A -85,B 0,C 180,E1 -15421.863,E2 -15421.863} C_VEL
LIN {X 0,Y 319.584,Z 605.675,A -85,B 0,C 180,E1 -15425.544,E2 -15425.544} C_VEL
LIN {X 0,Y 319.562,Z 605.678,A -85,B 0,C 180,E1 -15429.67,E2 -15429.67} C_VEL
LIN {X 0,Y 319.514,Z 605.682,A -85,B 0,C 180,E1 -15430.74,E2 -15430.74} C_VEL
LIN {X 0,Y 318.864,Z 605.768,A -85,B 0,C 180,E1 -15431.792,E2 -15431.792} C_VEL
LIN {X 0,Y 316.033,Z 606.123,A -85,B 0,C 180,E1 -15433.505,E2 -15433.505} C_VEL
LIN {X 0,Y 313.616,Z 606.42,A -85,B 0,C 180,E1 -15434.893,E2 -15434.893} C_VEL
LIN {X 0,Y 312.563,Z 606.548,A -85,B 0,C 180,E1 -15435.968,E2 -15435.968} C_VEL
LIN {X 0,Y 312.47,Z 606.557,A -85,B 0,C 180,E1 -15436.332,E2 -15436.332} C_VEL
LIN {X 0,Y 312.508,Z 606.554,A -85,B 0,C 180,E1 -15439.875,E2 -15439.875} C_VEL
LIN {X 0,Y 312.54,Z 606.55,A -85,B 0,C 180,E1 -15444.051,E2 -15444.051} C_VEL
LIN {X 0,Y 312.51,Z 606.556,A -85,B 0,C 180,E1 -15447.335,E2 -15447.335} C_VEL
LIN {X 0,Y 312.557,Z 606.55,A -85,B 0,C 180,E1 -15451.277,E2 -15451.277} C_VEL
LIN {X 0,Y 312.59,Z 606.544,A -85,B 0,C 180,E1 -15454.711,E2 -15454.711} C_VEL
LIN {X 0,Y 312.543,Z 606.549,A -85,B 0,C 180,E1 -15458.913,E2 -15458.913} C_VEL
LIN {X 0,Y 312.644,Z 606.54,A -85,B 0,C 180,E1 -15461.657,E2 -15461.657} C_VEL
LIN {X 0,Y 312.7,Z 606.532,A -85,B 0,C 180,E1 -15465.687,E2 -15465.687} C_VEL
LIN {X 0,Y 312.704,Z 606.532,A -85,B 0,C 180,E1 -15469.642,E2 -15469.642} C_VEL
LIN {X 0,Y 312.859,Z 606.514,A -85,B 0,C 180,E1 -15472.254,E2 -15472.254} C_VEL
LIN {X 0,Y 312.72,Z 606.528,A -85,B 0,C 180,E1 -15474.843,E2 -15474.843} C_VEL
LIN {X 0,Y 312.995,Z 606.494,A -85,B 0,C 180,E1 -15478.714,E2 -15478.714} C_VEL
LIN {X 0,Y 312.995,Z 606.492,A -85,B 0,C 180,E1 -15481.287,E2 -15481.287} C_VEL
LIN {X 0,Y 312.722,Z 606.527,A -85,B 0,C 180,E1 -15485.158,E2 -15485.158} C_VEL
LIN {X 0,Y 312.86,Z 606.511,A -85,B 0,C 180,E1 -15487.746,E2 -15487.746} C_VEL
LIN {X 0,Y 312.676,Z 606.534,A -85,B 0,C 180,E1 -15491.671,E2 -15491.671} C_VEL
LIN {X 0,Y 312.674,Z 606.535,A -85,B 0,C 180,E1 -15494.865,E2 -15494.865} C_VEL
LIN {X 0,Y 312.555,Z 606.549,A -85,B 0,C 180,E1 -15499.193,E2 -15499.193} C_VEL
LIN {X 0,Y 312.532,Z 606.555,A -85,B 0,C 180,E1 -15502.78,E2 -15502.78} C_VEL
LIN {X 0,Y 312.589,Z 606.55,A -85,B 0,C 180,E1 -15506.722,E2 -15506.722} C_VEL
LIN {X 0,Y 312.551,Z 606.549,A -85,B 0,C 180,E1 -15509.65,E2 -15509.65} C_VEL
LIN {X 0,Y 312.525,Z 606.552,A -85,B 0,C 180,E1 -15513.688,E2 -15513.688} C_VEL
LIN {X 0,Y 312.526,Z 606.554,A -85,B 0,C 180,E1 -15517.385,E2 -15517.385} C_VEL
LIN {X 0,Y 312.496,Z 606.56,A -85,B 0,C 180,E1 -15520.709,E2 -15520.709} C_VEL
LIN {X 0,Y 312.478,Z 606.558,A -85,B 0,C 180,E1 -15524.205,E2 -15524.205} C_VEL
LIN {X 0,Y 312.491,Z 606.557,A -85,B 0,C 180,E1 -15527.918,E2 -15527.918} C_VEL
LIN {X 0,Y 312.504,Z 606.559,A -85,B 0,C 180,E1 -15530.97,E2 -15530.97} C_VEL
LIN {X 0,Y 312.537,Z 606.551,A -85,B 0,C 180,E1 -15534.22,E2 -15534.22} C_VEL
LIN {X 0,Y 312.549,Z 606.657,A -85,B 0,C 180,E1 -15536.483,E2 -15536.483} C_VEL
LIN {X 0,Y 315.453,Z 620.135,A -85,B 0,C 180,E1 -15540.33,E2 -15540.33} C_VEL
LIN {X 0,Y 317.351,Z 629.932,A -85,B 0,C 180,E1 -15543.001,E2 -15543.001} C_VEL
LIN {X 0,Y 316.11,Z 640.102,A -85,B 0,C 180,E1 -15545.522,E2 -15545.522} C_VEL
LIN {X 0,Y 321.601,Z 682.741,A -85,B 0,C 180,E1 -15547.038,E2 -15547.038} C_VEL
LIN {X 0,Y 319.903,Z 748.924,A -85,B 0,C 180,E1 -15548.745,E2 -15548.745} C_VEL
LIN {X 0,Y 319.071,Z 763.027,A -85,B 0,C 180,E1 -15549.363,E2 -15549.363} C_VEL
LIN {X 0,Y 318.065,Z 775.178,A -85,B 0,C 180,E1 -15550.138,E2 -15550.138} C_VEL
LIN {X 0,Y 316.759,Z 787.787,A -85,B 0,C 180,E1 -15551.232,E2 -15551.232} C_VEL
LIN {X 0,Y 315.472,Z 799.097,A -85,B 0,C 180,E1 -15552.496,E2 -15552.496} C_VEL
LIN {X 0,Y 314.428,Z 809.085,A -85,B 0,C 180,E1 -15553.899,E2 -15553.899} C_VEL
LIN {X 0,Y 313.253,Z 819.408,A -85,B 0,C 180,E1 -15555.711,E2 -15555.711} C_VEL
LIN {X 0,Y 312.425,Z 826.893,A -85,B 0,C 180,E1 -15557.329,E2 -15557.329} C_VEL
LIN {X 0,Y 311.629,Z 834.23,A -85,B 0,C 180,E1 -15559.276,E2 -15559.276} C_VEL
LIN {X 0,Y 311.235,Z 839.169,A -85,B 0,C 180,E1 -15560.904,E2 -15560.904} C_VEL
LIN {X 0,Y 310.995,Z 843.936,A -85,B 0,C 180,E1 -15562.859,E2 -15562.859} C_VEL
LIN {X 0,Y 310.873,Z 847.522,A -85,B 0,C 180,E1 -15564.81,E2 -15564.81} C_VEL
LIN {X 0,Y 310.865,Z 849.309,A -85,B 0,C 180,E1 -15566.11,E2 -15566.11} C_VEL
LIN {X 0,Y 310.851,Z 850.635,A -85,B 0,C 180,E1 -15567.407,E2 -15567.407} C_VEL
LIN {X 0,Y 310.962,Z 851.55,A -85,B 0,C 180,E1 -15568.704,E2 -15568.704} C_VEL
LIN {X 0,Y 311.043,Z 852.039,A -85,B 0,C 180,E1 -15569.999,E2 -15569.999} C_VEL
LIN {X 0,Y 310.919,Z 852.051,A -85,B 0,C 180,E1 -15571.294,E2 -15571.294} C_VEL
LIN {X 0,Y 310.817,Z 851.655,A -85,B 0,C 180,E1 -15572.591,E2 -15572.591} C_VEL
LIN {X 0,Y 310.808,Z 850.86,A -85,B 0,C 180,E1 -15573.888,E2 -15573.888} C_VEL
LIN {X 0,Y 310.791,Z 848.97,A -85,B 0,C 180,E1 -15575.738,E2 -15575.738} C_VEL
LIN {X 0,Y 311.001,Z 845.85,A -85,B 0,C 180,E1 -15577.791,E2 -15577.791} C_VEL
LIN {X 0,Y 311.39,Z 841.801,A -85,B 0,C 180,E1 -15579.744,E2 -15579.744} C_VEL
LIN {X 0,Y 312.217,Z 835.638,A -85,B 0,C 180,E1 -15582.016,E2 -15582.016} C_VEL
LIN {X 0,Y 313.371,Z 828.876,A -85,B 0,C 180,E1 -15583.949,E2 -15583.949} C_VEL
LIN {X 0,Y 314.741,Z 820.5,A -85,B 0,C 180,E1 -15585.882,E2 -15585.882} C_VEL
LIN {X 0,Y 316.048,Z 812.096,A -85,B 0,C 180,E1 -15587.468,E2 -15587.468} C_VEL
LIN {X 0,Y 317.812,Z 801.82,A -85,B 0,C 180,E1 -15589.035,E2 -15589.035} C_VEL
LIN {X 0,Y 319.464,Z 791.714,A -85,B 0,C 180,E1 -15590.271,E2 -15590.271} C_VEL
LIN {X 0,Y 321.163,Z 779.101,A -85,B 0,C 180,E1 -15591.501,E2 -15591.501} C_VEL
LIN {X 0,Y 322.743,Z 766.712,A -85,B 0,C 180,E1 -15592.399,E2 -15592.399} C_VEL
LIN {X 0,Y 323.915,Z 753.982,A -85,B 0,C 180,E1 -15593.071,E2 -15593.071} C_VEL
LIN {X 0,Y 324.732,Z 739.906,A -85,B 0,C 180,E1 -15593.558,E2 -15593.558} C_VEL
LIN {X 0,Y 326.762,Z 683.29,A -85,B 0,C 180,E1 -15595.061,E2 -15595.061} C_VEL
LIN {X 0,Y 324.439,Z 664.494,A -85,B 0,C 180,E1 -15595.899,E2 -15595.899} C_VEL
LIN {X 0,Y 321.405,Z 647.523,A -85,B 0,C 180,E1 -15596.784,E2 -15596.784} C_VEL
LIN {X 0,Y 318.982,Z 636.282,A -85,B 0,C 180,E1 -15597.479,E2 -15597.479} C_VEL
LIN {X 0,Y 318.925,Z 633.836,A -85,B 0,C 180,E1 -15598.18,E2 -15598.18} C_VEL
LIN {X 0,Y 317.172,Z 624.874,A -85,B 0,C 180,E1 -15601.008,E2 -15601.008} C_VEL
LIN {X 0,Y 315.201,Z 616.503,A -85,B 0,C 180,E1 -15603.876,E2 -15603.876} C_VEL
LIN {X 0,Y 313.263,Z 609.243,A -85,B 0,C 180,E1 -15606.596,E2 -15606.596} C_VEL
LIN {X 0,Y 312.557,Z 606.553,A -85,B 0,C 180,E1 -15607.732,E2 -15607.732} C_VEL
LIN {X 0,Y 312.529,Z 606.56,A -85,B 0,C 180,E1 -15612.09,E2 -15612.09} C_VEL
LIN {X 0,Y 312.545,Z 606.556,A -85,B 0,C 180,E1 -15616.016,E2 -15616.016} C_VEL
LIN {X 0,Y 312.541,Z 606.555,A -85,B 0,C 180,E1 -15619.864,E2 -15619.864} C_VEL
LIN {X 0,Y 312.547,Z 606.552,A -85,B 0,C 180,E1 -15622.618,E2 -15622.618} C_VEL
LIN {X 0,Y 312.514,Z 606.552,A -85,B 0,C 180,E1 -15626.31,E2 -15626.31} C_VEL
LIN {X 0,Y 312.54,Z 606.55,A -85,B 0,C 180,E1 -15630.349,E2 -15630.349} C_VEL
LIN {X 0,Y 312.596,Z 606.54,A -85,B 0,C 180,E1 -15634.063,E2 -15634.063} C_VEL
LIN {X 0,Y 312.58,Z 606.546,A -85,B 0,C 180,E1 -15637.528,E2 -15637.528} C_VEL
LIN {X 0,Y 312.63,Z 606.542,A -85,B 0,C 180,E1 -15641.656,E2 -15641.656} C_VEL
LIN {X 0,Y 312.686,Z 606.532,A -85,B 0,C 180,E1 -15645.686,E2 -15645.686} C_VEL
LIN {X 0,Y 312.695,Z 606.534,A -85,B 0,C 180,E1 -15649.641,E2 -15649.641} C_VEL
LIN {X 0,Y 312.863,Z 606.512,A -85,B 0,C 180,E1 -15652.254,E2 -15652.254} C_VEL
LIN {X 0,Y 312.711,Z 606.53,A -85,B 0,C 180,E1 -15654.842,E2 -15654.842} C_VEL
LIN {X 0,Y 312.984,Z 606.497,A -85,B 0,C 180,E1 -15658.713,E2 -15658.713} C_VEL
LIN {X 0,Y 313.113,Z 606.484,A -85,B 0,C 180,E1 -15660,E2 -15660} C_VEL
LIN {X 0,Y 312.946,Z 606.505,A -85,B 0,C 180,E1 -15662.574,E2 -15662.574} C_VEL
LIN {X 0,Y 312.794,Z 606.649,A -85,B 0,C 180,E1 -15665.479,E2 -15665.479} C_VEL
LIN {X 0,Y 313.78,Z 610.042,A -85,B 0,C 180,E1 -15666.975,E2 -15666.975} C_VEL
LIN {X 0,Y 315.786,Z 613.649,A -85,B 0,C 180,E1 -15667.372,E2 -15667.372} C_VEL
LIN {X 0,Y 323.963,Z 629.997,A -85,B 0,C 180,E1 -15668.941,E2 -15668.941} C_VEL
LIN {X 0,Y 328.187,Z 640.012,A -85,B 0,C 180,E1 -15669.733,E2 -15669.733} C_VEL
LIN {X 0,Y 325.233,Z 715.292,A -85,B 0,C 180,E1 -15671.767,E2 -15671.767} C_VEL
LIN {X 0,Y 324.348,Z 728.968,A -85,B 0,C 180,E1 -15672.39,E2 -15672.39} C_VEL
LIN {X 0,Y 323.299,Z 741.42,A -85,B 0,C 180,E1 -15673.218,E2 -15673.218} C_VEL
LIN {X 0,Y 322.068,Z 752.685,A -85,B 0,C 180,E1 -15674.211,E2 -15674.211} C_VEL
LIN {X 0,Y 320.683,Z 763.08,A -85,B 0,C 180,E1 -15675.364,E2 -15675.364} C_VEL
LIN {X 0,Y 319.053,Z 773.537,A -85,B 0,C 180,E1 -15676.805,E2 -15676.805} C_VEL
LIN {X 0,Y 317.451,Z 782.752,A -85,B 0,C 180,E1 -15678.39,E2 -15678.39} C_VEL
LIN {X 0,Y 315.977,Z 790.687,A -85,B 0,C 180,E1 -15680.075,E2 -15680.075} C_VEL
LIN {X 0,Y 314.539,Z 797.93,A -85,B 0,C 180,E1 -15681.978,E2 -15681.978} C_VEL
LIN {X 0,Y 313.511,Z 803.439,A -85,B 0,C 180,E1 -15683.797,E2 -15683.797} C_VEL
LIN {X 0,Y 312.549,Z 808.488,A -85,B 0,C 180,E1 -15685.919,E2 -15685.919} C_VEL
LIN {X 0,Y 311.731,Z 812.721,A -85,B 0,C 180,E1 -15688.451,E2 -15688.451} C_VEL
LIN {X 0,Y 311.143,Z 815.226,A -85,B 0,C 180,E1 -15690.874,E2 -15690.874} C_VEL
LIN {X 0,Y 310.841,Z 816.23,A -85,B 0,C 180,E1 -15693.225,E2 -15693.225} C_VEL
LIN {X 0,Y 310.727,Z 815.918,A -85,B 0,C 180,E1 -15695.49,E2 -15695.49} C_VEL
LIN {X 0,Y 310.773,Z 814.435,A -85,B 0,C 180,E1 -15697.676,E2 -15697.676} C_VEL
LIN {X 0,Y 311.087,Z 811.816,A -85,B 0,C 180,E1 -15699.817,E2 -15699.817} C_VEL
LIN {X 0,Y 311.447,Z 808.151,A -85,B 0,C 180,E1 -15701.872,E2 -15701.872} C_VEL
LIN {X 0,Y 311.952,Z 803.388,A -85,B 0,C 180,E1 -15703.871,E2 -15703.871} C_VEL
LIN {X 0,Y 312.689,Z 796.831,A -85,B 0,C 180,E1 -15705.991,E2 -15705.991} C_VEL
LIN {X 0,Y 313.495,Z 790.076,A -85,B 0,C 180,E1 -15707.738,E2 -15707.738} C_VEL
LIN {X 0,Y 314.584,Z 781.095,A -85,B 0,C 180,E1 -15709.62,E2 -15709.62} C_VEL
LIN {X 0,Y 315.693,Z 771.849,A -85,B 0,C 180,E1 -15711.185,E2 -15711.185} C_VEL
LIN {X 0,Y 316.789,Z 762.013,A -85,B 0,C 180,E1 -15712.536,E2 -15712.536} C_VEL
LIN {X 0,Y 317.933,Z 750.092,A -85,B 0,C 180,E1 -15713.849,E2 -15713.849} C_VEL
LIN {X 0,Y 318.942,Z 738.311,A -85,B 0,C 180,E1 -15714.856,E2 -15714.856} C_VEL
LIN {X 0,Y 319.697,Z 725.405,A -85,B 0,C 180,E1 -15715.675,E2 -15715.675} C_VEL
LIN {X 0,Y 320.25,Z 711.704,A -85,B 0,C 180,E1 -15716.27,E2 -15716.27} C_VEL
LIN {X 0,Y 322.395,Z 634.032,A -85,B 0,C 180,E1 -15718.252,E2 -15718.252} C_VEL
LIN {X 0,Y 314.951,Z 613.09,A -85,B 0,C 180,E1 -15719.308,E2 -15719.308} C_VEL
LIN {X 0,Y 312.551,Z 606.552,A -85,B 0,C 180,E1 -15719.679,E2 -15719.679} C_VEL
LIN {X 0,Y 312.549,Z 606.55,A -85,B 0,C 180,E1 -15723.276,E2 -15723.276} C_VEL
LIN {X 0,Y 312.541,Z 606.556,A -85,B 0,C 180,E1 -15726.126,E2 -15726.126} C_VEL
LIN {X 0,Y 312.557,Z 606.549,A -85,B 0,C 180,E1 -15728.916,E2 -15728.916} C_VEL
LIN {X 0,Y 312.637,Z 606.539,A -85,B 0,C 180,E1 -15731.658,E2 -15731.658} C_VEL
LIN {X 0,Y 312.693,Z 606.532,A -85,B 0,C 180,E1 -15735.688,E2 -15735.688} C_VEL
LIN {X 0,Y 312.703,Z 606.53,A -85,B 0,C 180,E1 -15739.643,E2 -15739.643} C_VEL
LIN {X 0,Y 312.872,Z 606.513,A -85,B 0,C 180,E1 -15742.256,E2 -15742.256} C_VEL
LIN {X 0,Y 312.719,Z 606.53,A -85,B 0,C 180,E1 -15744.844,E2 -15744.844} C_VEL
LIN {X 0,Y 312.99,Z 606.498,A -85,B 0,C 180,E1 -15748.715,E2 -15748.715} C_VEL
LIN {X 0,Y 312.994,Z 606.494,A -85,B 0,C 180,E1 -15751.288,E2 -15751.288} C_VEL
LIN {X 0,Y 312.698,Z 606.531,A -85,B 0,C 180,E1 -15753.868,E2 -15753.868} C_VEL
LIN {X 0,Y 312.912,Z 606.508,A -85,B 0,C 180,E1 -15756.449,E2 -15756.449} C_VEL
LIN {X 0,Y 312.789,Z 606.522,A -85,B 0,C 180,E1 -15759.05,E2 -15759.05} C_VEL
LIN {X 0,Y 312.637,Z 606.542,A -85,B 0,C 180,E1 -15762.992,E2 -15762.992} C_VEL
LIN {X 0,Y 312.641,Z 606.538,A -85,B 0,C 180,E1 -15765.651,E2 -15765.651} C_VEL
LIN {X 0,Y 312.633,Z 606.54,A -85,B 0,C 180,E1 -15769.237,E2 -15769.237} C_VEL
LIN {X 0,Y 312.549,Z 606.553,A -85,B 0,C 180,E1 -15772.791,E2 -15772.791} C_VEL
LIN {X 0,Y 312.6,Z 606.543,A -85,B 0,C 180,E1 -15775.934,E2 -15775.934} C_VEL
LIN {X 0,Y 312.542,Z 606.551,A -85,B 0,C 180,E1 -15779.652,E2 -15779.652} C_VEL
LIN {X 0,Y 312.523,Z 606.551,A -85,B 0,C 180,E1 -15783.69,E2 -15783.69} C_VEL
LIN {X 0,Y 312.524,Z 606.556,A -85,B 0,C 180,E1 -15787.387,E2 -15787.387} C_VEL
LIN {X 0,Y 312.493,Z 606.557,A -85,B 0,C 180,E1 -15790.724,E2 -15790.724} C_VEL
LIN {X 0,Y 312.476,Z 606.558,A -85,B 0,C 180,E1 -15794.207,E2 -15794.207} C_VEL
LIN {X 0,Y 312.47,Z 606.557,A -85,B 0,C 180,E1 -15796.332,E2 -15796.332} C_VEL
LIN {X 0,Y 311.793,Z 606.648,A -85,B 0,C 180,E1 -15797.408,E2 -15797.408} C_VEL
LIN {X 0,Y 308.972,Z 606.996,A -85,B 0,C 180,E1 -15799.161,E2 -15799.161} C_VEL
LIN {X 0,Y 306.583,Z 607.294,A -85,B 0,C 180,E1 -15800.582,E2 -15800.582} C_VEL
LIN {X 0,Y 305.546,Z 607.421,A -85,B 0,C 180,E1 -15801.682,E2 -15801.682} C_VEL
LIN {X 0,Y 305.454,Z 607.429,A -85,B 0,C 180,E1 -15802.054,E2 -15802.054} C_VEL
LIN {X 0,Y 305.47,Z 607.432,A -85,B 0,C 180,E1 -15805.922,E2 -15805.922} C_VEL
LIN {X 0,Y 305.469,Z 607.436,A -85,B 0,C 180,E1 -15809.592,E2 -15809.592} C_VEL
LIN {X 0,Y 305.526,Z 607.424,A -85,B 0,C 180,E1 -15812.609,E2 -15812.609} C_VEL
LIN {X 0,Y 305.51,Z 607.43,A -85,B 0,C 180,E1 -15815.539,E2 -15815.539} C_VEL
LIN {X 0,Y 305.512,Z 607.429,A -85,B 0,C 180,E1 -15819.815,E2 -15819.815} C_VEL
LIN {X 0,Y 305.58,Z 607.414,A -85,B 0,C 180,E1 -15822.603,E2 -15822.603} C_VEL
LIN {X 0,Y 305.655,Z 607.406,A -85,B 0,C 180,E1 -15825.349,E2 -15825.349} C_VEL
LIN {X 0,Y 305.641,Z 607.41,A -85,B 0,C 180,E1 -15829.4,E2 -15829.4} C_VEL
LIN {X 0,Y 305.803,Z 607.395,A -85,B 0,C 180,E1 -15832.074,E2 -15832.074} C_VEL
LIN {X 0,Y 305.691,Z 607.404,A -85,B 0,C 180,E1 -15834.724,E2 -15834.724} C_VEL
LIN {X 0,Y 305.961,Z 607.37,A -85,B 0,C 180,E1 -15838.684,E2 -15838.684} C_VEL
LIN {X 0,Y 305.962,Z 607.367,A -85,B 0,C 180,E1 -15841.316,E2 -15841.316} C_VEL
LIN {X 0,Y 305.693,Z 607.402,A -85,B 0,C 180,E1 -15845.277,E2 -15845.277} C_VEL
LIN {X 0,Y 305.804,Z 607.391,A -85,B 0,C 180,E1 -15847.926,E2 -15847.926} C_VEL
LIN {X 0,Y 305.61,Z 607.415,A -85,B 0,C 180,E1 -15851.945,E2 -15851.945} C_VEL
LIN {X 0,Y 305.615,Z 607.413,A -85,B 0,C 180,E1 -15855.014,E2 -15855.014} C_VEL
LIN {X 0,Y 305.524,Z 607.428,A -85,B 0,C 180,E1 -15858.787,E2 -15858.787} C_VEL
LIN {X 0,Y 305.492,Z 607.43,A -85,B 0,C 180,E1 -15863.039,E2 -15863.039} C_VEL
LIN {X 0,Y 305.56,Z 607.421,A -85,B 0,C 180,E1 -15866.229,E2 -15866.229} C_VEL
LIN {X 0,Y 305.502,Z 607.43,A -85,B 0,C 180,E1 -15869.05,E2 -15869.05} C_VEL
LIN {X 0,Y 305.471,Z 607.431,A -85,B 0,C 180,E1 -15873.516,E2 -15873.516} C_VEL
LIN {X 0,Y 305.478,Z 607.435,A -85,B 0,C 180,E1 -15876.739,E2 -15876.739} C_VEL
LIN {X 0,Y 305.46,Z 607.435,A -85,B 0,C 180,E1 -15880.599,E2 -15880.599} C_VEL
LIN {X 0,Y 305.424,Z 607.439,A -85,B 0,C 180,E1 -15884.492,E2 -15884.492} C_VEL
LIN {X 0,Y 305.447,Z 607.434,A -85,B 0,C 180,E1 -15888.143,E2 -15888.143} C_VEL
LIN {X 0,Y 305.473,Z 607.433,A -85,B 0,C 180,E1 -15891.596,E2 -15891.596} C_VEL
LIN {X 0,Y 305.468,Z 607.435,A -85,B 0,C 180,E1 -15894.886,E2 -15894.886} C_VEL
LIN {X 0,Y 305.505,Z 607.547,A -85,B 0,C 180,E1 -15896.123,E2 -15896.123} C_VEL
LIN {X 0,Y 308.346,Z 620.842,A -85,B 0,C 180,E1 -15900.011,E2 -15900.011} C_VEL
LIN {X 0,Y 310.257,Z 630.184,A -85,B 0,C 180,E1 -15902.63,E2 -15902.63} C_VEL
LIN {X 0,Y 310.153,Z 633.198,A -85,B 0,C 180,E1 -15903.413,E2 -15903.413} C_VEL
LIN {X 0,Y 309.277,Z 639.694,A -85,B 0,C 180,E1 -15905.059,E2 -15905.059} C_VEL
LIN {X 0,Y 314.878,Z 684.357,A -85,B 0,C 180,E1 -15906.683,E2 -15906.683} C_VEL
LIN {X 0,Y 313.097,Z 748.744,A -85,B 0,C 180,E1 -15908.39,E2 -15908.39} C_VEL
LIN {X 0,Y 312.228,Z 762.739,A -85,B 0,C 180,E1 -15909.019,E2 -15909.019} C_VEL
LIN {X 0,Y 311.158,Z 775.355,A -85,B 0,C 180,E1 -15909.851,E2 -15909.851} C_VEL
LIN {X 0,Y 309.811,Z 787.824,A -85,B 0,C 180,E1 -15910.967,E2 -15910.967} C_VEL
LIN {X 0,Y 308.506,Z 799.056,A -85,B 0,C 180,E1 -15912.259,E2 -15912.259} C_VEL
LIN {X 0,Y 307.399,Z 809.22,A -85,B 0,C 180,E1 -15913.735,E2 -15913.735} C_VEL
LIN {X 0,Y 306.345,Z 818.416,A -85,B 0,C 180,E1 -15915.382,E2 -15915.382} C_VEL
LIN {X 0,Y 305.291,Z 827.381,A -85,B 0,C 180,E1 -15917.366,E2 -15917.366} C_VEL
LIN {X 0,Y 304.527,Z 834.504,A -85,B 0,C 180,E1 -15919.359,E2 -15919.359} C_VEL
LIN {X 0,Y 304.076,Z 840.182,A -85,B 0,C 180,E1 -15921.358,E2 -15921.358} C_VEL
LIN {X 0,Y 303.85,Z 844.602,A -85,B 0,C 180,E1 -15923.358,E2 -15923.358} C_VEL
